DATA_BLOCK "ZEN_Bef"
{ S7_Optimized_Access := 'FALSE' }
VERSION : 0.1
NON_RETAIN
   STRUCT
      ZEN_Quit_BF : Bool;   // UV BG - SPS Quit
      ZEN_Bed_Sperre_BF : Bool;   // UV BG Bedienstelle - Bedienung sperren
      ZEN_Bed_Frg_BF : Bool;   // UV BG Bedienstelle - Bedienung freigeben
      ZEN_ObjS_unscharf_BF : Bool;   // Betriebsgebäude - Objektschutz - Freischaltung
      ZEN_ObjS_scharf_BF : Bool;   // Betriebsgebäude - Objektschutz - Scharfschaltung
      ZEN_GWA_RST_BF : Bool;   // Gaswarnanlagen - Fern-Reset
      ZEN_IEC_RST_BF : Bool;   // IEC-Stack Reset
      ZEN_Res_DB101_0_7 : Bool;   // Reserve
      Biocos1_BA_SU_BF : Bool;   // Steuerung Biocos 1 - Betriebsart - Schaltuhrbetrieb - Befehl
      Biocos1_BA_P1_BF : Bool;   // Steuerung Biocos 1 - Betriebsart - Parametersatz 1 - Befehl
      Biocos1_BA_P2_BF : Bool;   // Steuerung Biocos 1 - Betriebsart - Parametersatz 2 - Befehl
      Biocos1_BA_Aus_BF : Bool;   // Steuerung Biocos 1 - Betriebsart - Aus - Befehl
      Biocos1_Auto_Bel_O2_Ein_BF : Bool;   // Steuerung Biocos 1 - Automatik - Belüftung nach O2-Gehalt - Befehl Ein
      Biocos1_Auto_Bel_O2_Aus_BF : Bool;   // Steuerung Biocos 1 - Automatik - Belüftung nach O2-Gehalt - Befehl Aus
      Biocos1_Auto_UeSS_Menge_Ein_BF : Bool;   // Steuerung Biocos 1 - Automatik - ÜSS-Abzug nach Menge - Befehl Ein
      Biocos1_Auto_UeSS_Menge_Aus_BF : Bool;   // Steuerung Biocos 1 - Automatik - ÜSS-Abzug nach Menge - Befehl Aus
      Biocos2_BA_SU_BF : Bool;   // Steuerung Biocos 2 - Betriebsart - Schaltuhrbetrieb - Befehl
      Biocos2_BA_P1_BF : Bool;   // Steuerung Biocos 2 - Betriebsart - Parametersatz 1 - Befehl
      Biocos2_BA_P2_BF : Bool;   // Steuerung Biocos 2 - Betriebsart - Parametersatz 2 - Befehl
      Biocos2_BA_Aus_BF : Bool;   // Steuerung Biocos 2 - Betriebsart - Aus - Befehl
      Biocos2_Auto_Bel_O2_Ein_BF : Bool;   // Steuerung Biocos 2 - Automatik - Belüftung nach O2-Gehalt - Befehl Ein
      Biocos2_Auto_Bel_O2_Aus_BF : Bool;   // Steuerung Biocos 2 - Automatik - Belüftung nach O2-Gehalt - Befehl Aus
      Biocos2_Auto_UeSS_Menge_Ein_BF : Bool;   // Steuerung Biocos 2 - Automatik - ÜSS-Abzug nach Menge - Befehl Ein
      Biocos2_Auto_UeSS_Menge_Aus_BF : Bool;   // Steuerung Biocos 2 - Automatik - ÜSS-Abzug nach Menge - Befehl Aus
      Zulauf_PW_BA_Auto_BF : Bool;   // Steuerung Zulauf/Freigabe Pumpwerke - Betriebsart - Automatik - Befehl
      Zulauf_PW_BA_Aus_BF : Bool;   // Steuerung Zulauf/Freigabe Pumpwerke - Betriebsart - Aus - Befehl
      Zulauf_PW_BA_EFrg_Ein_BF : Bool;   // Steuerung Zulauf/Freigabe Pumpwerke - Betriebsart - einzelne Freigabe zuschalten - Befehl
      Zulauf_PW_BA_EFrg_Aus_BF : Bool;   // Steuerung Zulauf/Freigabe Pumpwerke - Betriebsart - einzelne Freigabe abschalten - Befehl
      Zulauf_PW_BA_SFrg_Ein_BF : Bool;   // Steuerung Zulauf/Freigabe Pumpwerke - Betriebsart - alle Freigaben zuschalten - Befehl
      Zulauf_PW_BA_SFrg_Aus_BF : Bool;   // Steuerung Zulauf/Freigabe Pumpwerke - Betriebsart - alle Freigaben abschalten - Befehl
      ZEN_Res_DB101_3_6 : Bool;   // Reserve
      ZEN_Res_DB101_3_7 : Bool;   // Reserve
      Schlamm_TW_BA_Auto_BF : Bool;   // Steuerung Trübwasserpumpwerk - Betriebsart - Automatik - Befehl
      Schlamm_TW_BA_Aus_BF : Bool;   // Steuerung Trübwasserpumpwerk - Betriebsart - Aus - Befehl
      ZEN_Res_DB101_4_2 : Bool;   // Reserve
      ZEN_Res_DB101_4_3 : Bool;   // Reserve
      ZEN_Res_DB101_4_4 : Bool;   // Reserve
      ZEN_Res_DB101_4_5 : Bool;   // Reserve
      ZEN_Res_DB101_4_6 : Bool;   // Reserve
      ZEN_Res_DB101_4_7 : Bool;   // Reserve
      Schlamm_Besch_BA_Auto_BF : Bool;   // Steuerung Beschickung Schlammbeete - Betriebsart - Automatik - Befehl
      Schlamm_Besch_BA_Aus_BF : Bool;   // Steuerung Beschickung Schlammbeete - Betriebsart - Aus - Befehl
      ZEN_Res_DB101_5_2 : Bool;   // Reserve
      ZEN_Res_DB101_5_3 : Bool;   // Reserve
      ZEN_Res_DB101_5_4 : Bool;   // Reserve
      ZEN_Res_DB101_5_5 : Bool;   // Reserve
      ZEN_Res_DB101_5_6 : Bool;   // Reserve
      ZEN_Res_DB101_5_7 : Bool;   // Reserve
      PO4_Elim_BA_Auto_BF : Bool;   // Steuerung PO4-Elimination - Betriebsart - Automatik - Befehl
      PO4_Elim_BA_Hand_BF : Bool;   // Steuerung PO4-Elimination - Betriebsart - Handvorgabe - Befehl
      PO4_Elim_BA_Aus_BF : Bool;   // Steuerung PO4-Elimination - Betriebsart - Aus - Befehl
      PO4_Elim_DF_RST_BF : Bool;   // Steuerung PO4-Elimination - Menge Fällmittel - Reset - Befehl
      ZEN_Res_DB101_6_4 : Bool;   // Reserve
      ZEN_Res_DB101_6_5 : Bool;   // Reserve
      ZEN_Res_DB101_6_6 : Bool;   // Reserve
      ZEN_Res_DB101_6_7 : Bool;   // Reserve
      Biocos1_BA_O2_Reg_FW_BF : Bool;   // Steuerung Biocos 1 - Betriebsart O2-Regler - Festwert - Befehl
      Biocos1_BA_O2_Reg_Auto_BF : Bool;   // Steuerung Biocos 1 - Betriebsart O2-Regler - Automatik - Befehl
      ZEN_Res_DB101_7_2 : Bool;   // Reserve
      ZEN_Res_DB101_7_3 : Bool;   // Reserve
      ZEN_Res_DB101_7_4 : Bool;   // Reserve
      ZEN_Res_DB101_7_5 : Bool;   // Reserve
      ZEN_Res_DB101_7_6 : Bool;   // Reserve
      ZEN_Res_DB101_7_7 : Bool;   // Reserve
      Biocos2_BA_O2_Reg_FW_BF : Bool;   // Steuerung Biocos 2 - Betriebsart O2-Regler - Festwert - Befehl
      Biocos2_BA_O2_Reg_Auto_BF : Bool;   // Steuerung Biocos 2 - Betriebsart O2-Regler - Automatik - Befehl
      ZEN_Res_DB101_8_2 : Bool;   // Reserve
      ZEN_Res_DB101_8_3 : Bool;   // Reserve
      ZEN_Res_DB101_8_4 : Bool;   // Reserve
      ZEN_Res_DB101_8_5 : Bool;   // Reserve
      ZEN_Res_DB101_8_6 : Bool;   // Reserve
      ZEN_Res_DB101_8_7 : Bool;   // Reserve
      RES : Array[0..9] of Byte;
   END_STRUCT;


BEGIN

END_DATA_BLOCK

DATA_BLOCK "IDB_SL_Org_ASDU_1"
{ S7_Optimized_Access := 'FALSE' }
AUTHOR : SIE_GST
FAMILY : S7_IEC
VERSION : 0.1
"SL_Org_Asdu_1"

BEGIN

END_DATA_BLOCK

DATA_BLOCK "IDB_MA_Org_ASDU_1"
{ S7_Optimized_Access := 'FALSE' }
AUTHOR : SIE_GST
FAMILY : S7_IEC
VERSION : 0.1
"MA_Org_Asdu_n"

BEGIN

END_DATA_BLOCK

DATA_BLOCK "DB_IEC_PW_Image"
{ S7_Optimized_Access := 'FALSE' }
VERSION : 0.1
   STRUCT
      FW_APW_Oeb_KB : "T_IEC_PW_Image";   // Oebisfelde APW Krumme Breite
      FW_APW_BrR_DM : "T_IEC_PW_Image";   // Breitenrode APW Denkmal
      FW_APW_Oeb_Tu : "T_IEC_PW_Image";   // Oebisfelde APW Tunnel
      FW_APW_Oeb_KS : "T_IEC_PW_Image";   // Oebisfelde APW Klötzer Str.
      FW_APW_Oeb_PG : "T_IEC_PW_Image";   // Oebisfelde APW Papengraben
      FW_APW_Oeb_LW : "T_IEC_PW_Image";   // Oebisfelde APW Lehmweg
      FW_APW_GeD_WG : "T_IEC_PW_Image";   // Gehrendorf APW Wiesengrund
      FW_APW_GeD_AA : "T_IEC_PW_Image";   // Gehrendorf APW An der Aller
      FW_APW_WaD : "T_IEC_PW_Image";   // Wassensdorf APW
      FW_APW_WeD : "T_IEC_PW_Image";   // Weddendorf APW
      FW_APW_NiD : "T_IEC_PW_Image";   // Niendorf APW
      FW_APW_LoS : "T_IEC_PW_Image";   // Lockstedt APW
      FW_APW_Oeb_Ge : "T_IEC_PW_Image";   // Oebisfelde APW Gewerbe
      FW_APW_BuH : "T_IEC_PW_Image";   // Buchhorst APW
      FW_APW_BrR_TS : "T_IEC_PW_Image";   // Breitenrode APW Trafostation
   END_STRUCT;


BEGIN

END_DATA_BLOCK

DATA_BLOCK "ZEN_SW"
{ S7_Optimized_Access := 'FALSE' }
VERSION : 0.1
   STRUCT
      BB_Auto_GeblW_ZZ_SW : DInt;   // Steuerung Belüftung - Automatik - Zykluszeit Gebläsetausch
      Biocos1_Auto_Bel_O2_Int_SW : Real;   // Steuerung Biocos 1 - Automatik - Sollwert O2-Gehalt am Ende Belüftungsintervall
      Biocos1_Auto_Bel_O2_min_SW : Real;   // Steuerung Biocos 1 - Automatik - Grenzwert Sauerstoffeintrag min. pro Belüftungsphase
      Biocos1_Auto_Bel_O2_Zt_min_SW : DInt;   // Steuerung Biocos 1 - Automatik - Mindestbelüftungsdauer pro Intervall
      Biocos1_Auto_UeSS_Zyk_SW : DInt;   // Steuerung Biocos 1 - Automatik - ÜSS-Abzug alle X Zyklen
      Biocos1_Auto_P1_Start_SW : DInt;   // Steuerung Biocos 1 - Automatik - Startzeit Parametersatz 1
      Biocos1_Auto_P2_Start_SW : DInt;   // Steuerung Biocos 1 - Automatik - Startzeit Parametersatz 2
      Biocos1_Auto_U_Zt_P1_SW : DInt;   // Steuerung Biocos 1 - Automatik - Sollwert U-Phase - Parametersatz 1
      Biocos1_Auto_V_Zt_P1_SW : DInt;   // Steuerung Biocos 1 - Automatik - Sollwert V-Phase - Parametersatz 1
      Biocos1_Auto_Bel_Vz_P1_SW : DInt;   // Steuerung Biocos 1 - Automatik - Sollwert Verzögerungszeit Belüftungsphase - Parametersatz 1
      Biocos1_Auto_Bel_Int_P1_SW : DInt;   // Steuerung Biocos 1 - Automatik - Sollwert Anzahl Belüftungsintervalle - Parametersatz 1
      Biocos1_Auto_Bel_Int_Zt_P1_SW : DInt;   // Steuerung Biocos 1 - Automatik - Sollwert Belüftungsdauer (fest) pro Intervall - Parametersatz 1
      Biocos1_Auto_UeSS_Zt_P1_SW : DInt;   // Steuerung Biocos 1 - Automatik - Sollwert ÜSS-Abzug Dauer - Parametersatz 1
      Biocos1_Auto_UeSS_Df_P1_SW : Real;   // Steuerung Biocos 1 - Automatik - Sollwert ÜSS-Abzug Menge - Parametersatz 1
      Biocos1_Auto_SR1_Zt_P1_SW : DInt;   // Steuerung Biocos 1 - Automatik - Sollwert Dauer Schlammrückführung SU-Becken 1 - Parametersatz 1
      Biocos1_Auto_SR2_Zt_P1_SW : DInt;   // Steuerung Biocos 1 - Automatik - Sollwert Dauer Schlammrückführung SU-Becken 2 - Parametersatz 1
      Biocos1_Auto_U_Zt_P2_SW : DInt;   // Steuerung Biocos 1 - Automatik - Sollwert U-Phase - Parametersatz 2
      Biocos1_Auto_V_Zt_P2_SW : DInt;   // Steuerung Biocos 1 - Automatik - Sollwert V-Phase - Parametersatz 2
      Biocos1_Auto_Bel_Vz_P2_SW : DInt;   // Steuerung Biocos 1 - Automatik - Sollwert Verzögerungszeit Belüftungsphase - Parametersatz 2
      Biocos1_Auto_Bel_Int_P2_SW : DInt;   // Steuerung Biocos 1 - Automatik - Sollwert Anzahl Belüftungsintervalle - Parametersatz 2
      Biocos1_Auto_Bel_Int_Zt_P2_SW : DInt;   // Steuerung Biocos 1 - Automatik - Sollwert Belüftungsdauer (fest) pro Intervall - Parametersatz 2
      Biocos1_Auto_UeSS_Zt_P2_SW : DInt;   // Steuerung Biocos 1 - Automatik - Sollwert ÜSS-Abzug Dauer - Parametersatz 2
      Biocos1_Auto_UeSS_Df_P2_SW : Real;   // Steuerung Biocos 1 - Automatik - Sollwert ÜSS-Abzug Menge - Parametersatz 2
      Biocos1_Auto_SR1_Zt_P2_SW : DInt;   // Steuerung Biocos 1 - Automatik - Sollwert Dauer Schlammrückführung SU-Becken 1 - Parametersatz 2
      Biocos1_Auto_SR2_Zt_P2_SW : DInt;   // Steuerung Biocos 1 - Automatik - Sollwert Dauer Schlammrückführung SU-Becken 2 - Parametersatz 2
      Biocos2_Auto_Bel_O2_Int_SW : Real;   // Steuerung Biocos 2 - Automatik - Sollwert O2-Gehalt am Ende Belüftungsintervall
      Biocos2_Auto_Bel_O2_min_SW : Real;   // Steuerung Biocos 2 - Automatik - Grenzwert Sauerstoffeintrag min. pro Belüftungsphase
      Biocos2_Auto_Bel_O2_Zt_min_SW : DInt;   // Steuerung Biocos 2 - Automatik - Mindestbelüftungsdauer pro Intervall
      Biocos2_Auto_UeSS_Zyk_SW : DInt;   // Steuerung Biocos 2 - Automatik - ÜSS-Abzug alle X Zyklen
      Biocos2_Auto_P1_Start_SW : DInt;   // Steuerung Biocos 2 - Automatik - Startzeit Parametersatz 1
      Biocos2_Auto_P2_Start_SW : DInt;   // Steuerung Biocos 2 - Automatik - Startzeit Parametersatz 2
      Biocos2_Auto_U_Zt_P1_SW : DInt;   // Steuerung Biocos 2 - Automatik - Sollwert U-Phase - Parametersatz 1
      Biocos2_Auto_V_Zt_P1_SW : DInt;   // Steuerung Biocos 2 - Automatik - Sollwert V-Phase - Parametersatz 1
      Biocos2_Auto_Bel_Vz_P1_SW : DInt;   // Steuerung Biocos 2 - Automatik - Sollwert Verzögerungszeit Belüftungsphase - Parametersatz 1
      Biocos2_Auto_Bel_Int_P1_SW : DInt;   // Steuerung Biocos 2 - Automatik - Sollwert Anzahl Belüftungsintervalle - Parametersatz 1
      Biocos2_Auto_Bel_Int_Zt_P1_SW : DInt;   // Steuerung Biocos 2 - Automatik - Sollwert Belüftungsdauer (fest) pro Intervall - Parametersatz 1
      Biocos2_Auto_UeSS_Zt_P1_SW : DInt;   // Steuerung Biocos 2 - Automatik - Sollwert ÜSS-Abzug Dauer - Parametersatz 1
      Biocos2_Auto_UeSS_Df_P1_SW : Real;   // Steuerung Biocos 2 - Automatik - Sollwert ÜSS-Abzug Menge - Parametersatz 1
      Biocos2_Auto_SR1_Zt_P1_SW : DInt;   // Steuerung Biocos 2 - Automatik - Sollwert Dauer Schlammrückführung SU-Becken 1 - Parametersatz 1
      Biocos2_Auto_SR2_Zt_P1_SW : DInt;   // Steuerung Biocos 2 - Automatik - Sollwert Dauer Schlammrückführung SU-Becken 2 - Parametersatz 1
      Biocos2_Auto_U_Zt_P2_SW : DInt;   // Steuerung Biocos 2 - Automatik - Sollwert U-Phase - Parametersatz 2
      Biocos2_Auto_V_Zt_P2_SW : DInt;   // Steuerung Biocos 2 - Automatik - Sollwert V-Phase - Parametersatz 2
      Biocos2_Auto_Bel_Vz_P2_SW : DInt;   // Steuerung Biocos 2 - Automatik - Sollwert Verzögerungszeit Belüftungsphase - Parametersatz 2
      Biocos2_Auto_Bel_Int_P2_SW : DInt;   // Steuerung Biocos 2 - Automatik - Sollwert Anzahl Belüftungsintervalle - Parametersatz 2
      Biocos2_Auto_Bel_Int_Zt_P2_SW : DInt;   // Steuerung Biocos 2 - Automatik - Sollwert Belüftungsdauer (fest) pro Intervall - Parametersatz 2
      Biocos2_Auto_UeSS_Zt_P2_SW : DInt;   // Steuerung Biocos 2 - Automatik - Sollwert ÜSS-Abzug Dauer - Parametersatz 2
      Biocos2_Auto_UeSS_Df_P2_SW : Real;   // Steuerung Biocos 2 - Automatik - Sollwert ÜSS-Abzug Menge - Parametersatz 2
      Biocos2_Auto_SR1_Zt_P2_SW : DInt;   // Steuerung Biocos 2 - Automatik - Sollwert Dauer Schlammrückführung SU-Becken 1 - Parametersatz 2
      Biocos2_Auto_SR2_Zt_P2_SW : DInt;   // Steuerung Biocos 2 - Automatik - Sollwert Dauer Schlammrückführung SU-Becken 2 - Parametersatz 2
      Zulauf_PW_Auto_DF_max_SW : Real;   // Steuerung Zulauf/Freigabe Pumpwerke - Grenzwert max. Durchflußmenge durch die KA
      Zulauf_PW_Auto_Niv_max_SW : Real;   // Steuerung Zulauf/Freigabe Pumpwerke - Niveau Vorlageschacht Zulauf - alle Freigaben ext. PW abschalten
      Zulauf_PW_Auto_Niv_AS_SW : Real;   // Steuerung Zulauf/Freigabe Pumpwerke - Niveau Vorlageschacht Zulauf - Freigabe ext. PW abschalten
      Zulauf_PW_Auto_Niv_ZS_SW : Real;   // Steuerung Zulauf/Freigabe Pumpwerke - Niveau Vorlageschacht Zulauf - Freigabe ext. PW zuschalten
      Zulauf_PW_Auto_Niv_min_SW : Real;   // Steuerung Zulauf/Freigabe Pumpwerke - Niveau Vorlageschacht Zulauf - alle Freigaben ext. PW zuschalten
      Zulauf_PW_Auto_Zyk_SW : DInt;   // Steuerung Zulauf/Freigabe Pumpwerke - Zykluszeit Zu-/Abschaltung Pumpwerke
      Schlamm_TW_Auto_Frg_Zt_Ein_SW : DInt;   // Steuerung Trübwasserpumpwerk - Startzeit Freigabe Abzug
      Schlamm_TW_Auto_Frg_Zt_Aus_SW : DInt;   // Steuerung Trübwasserpumpwerk - Endzeit Freigabe Abzug
      Schlamm_TW_Auto_Niv_2P_Ein_SW : Real;   // Steuerung Trübwasserpumpwerk - Niveau Trübwasserschacht - Abpumpen 2 Pumpen Ein
      Schlamm_TW_Auto_Niv_1P_Ein_SW : Real;   // Steuerung Trübwasserpumpwerk - Niveau Trübwasserschacht - Abpumpen 1 Pumpe Ein
      Schlamm_TW_Auto_Niv_Aus_SW : Real;   // Steuerung Trübwasserpumpwerk - Niveau Trübwasserschacht - Abpumpen Aus
      Schlamm_Besch_Auto_Menge_SW : DInt;   // Steuerung Beschickung Schlammbeete - Menge Beschickung - Sollwert
      Schlamm_Besch_Auto_Zt_max_SW : DInt;   // Steuerung Beschickung Schlammbeete - Überwachungszeit
      PO4_Elim_BA_Hand_SW : Real;   // Steuerung PO4-Elimination - Betriebsart Hand - Menge Fällmittel - Sollwert
      Biocos1_Auto_Bel_O2_Reg_FW : Real;   // Steuerung Biocos 1 - Automatik O2-Regler - Vorgabe Festwert Blockdrehzahl für Ansteuerung Gebläse
      Biocos1_Auto_Bel_O2_Reg_GW_max : Real;   // Steuerung Biocos 1 - Automatik O2-Regler - Sollwert O2-Gehalt max -> Abschaltung Gebläse
      Biocos1_Auto_Bel_O2_Reg_GW_ein : Real;   // Steuerung Biocos 1 - Automatik O2-Regler - Sollwert O2-Gehalt min -> Einschaltung Gebläse
      Biocos1_Auto_Bel_O2_Reg_SW_max : Real;   // Steuerung Biocos 1 - Automatik O2-Regler - Sollwert O2-Gehalt max -> Gebläse auf min-Drehzahl
      Biocos1_Auto_Bel_O2_Reg_SW_min : Real;   // Steuerung Biocos 1 - Automatik O2-Regler - Sollwert O2-Gehalt min -> Gebläse auf max-Drehzahl
      Biocos1_Auto_Bel_O2_Reg_DZ_max : Real;   // Steuerung Biocos 1 - Automatik O2-Regler - Sollwert Blockdrehzahl max bei O2 min
      Biocos1_Auto_Bel_O2_Reg_DZ_min : Real;   // Steuerung Biocos 1 - Automatik O2-Regler - Sollwert Blockdrehzahl min bei O2 max
      Biocos2_Auto_Bel_O2_Reg_FW : Real;   // Steuerung Biocos 2 - Automatik O2-Regler - Vorgabe Festwert Blockdrehzahl für Ansteuerung Gebläse
      Biocos2_Auto_Bel_O2_Reg_GW_max : Real;   // Steuerung Biocos 2 - Automatik O2-Regler - Sollwert O2-Gehalt max -> Abschaltung Gebläse
      Biocos2_Auto_Bel_O2_Reg_GW_ein : Real;   // Steuerung Biocos 2 - Automatik O2-Regler - Sollwert O2-Gehalt min -> Einschaltung Gebläse
      Biocos2_Auto_Bel_O2_Reg_SW_max : Real;   // Steuerung Biocos 2 - Automatik O2-Regler - Sollwert O2-Gehalt max -> Gebläse auf min-Drehzahl
      Biocos2_Auto_Bel_O2_Reg_SW_min : Real;   // Steuerung Biocos 2 - Automatik O2-Regler - Sollwert O2-Gehalt min -> Gebläse auf max-Drehzahl
      Biocos2_Auto_Bel_O2_Reg_DZ_max : Real;   // Steuerung Biocos 2 - Automatik O2-Regler - Sollwert Blockdrehzahl max bei O2 min
      Biocos2_Auto_Bel_O2_Reg_DZ_min : Real;   // Steuerung Biocos 2 - Automatik O2-Regler - Sollwert Blockdrehzahl min bei O2 max
      RES : Array[0..9] of Byte;
   END_STRUCT;


BEGIN
   BB_Auto_GeblW_ZZ_SW := 24;
   Biocos1_Auto_Bel_O2_Int_SW := 2.0;
   Biocos1_Auto_Bel_O2_min_SW := 0.5;
   Biocos1_Auto_Bel_O2_Zt_min_SW := 300;
   Biocos1_Auto_UeSS_Zyk_SW := 1;
   Biocos1_Auto_P1_Start_SW := 8;
   Biocos1_Auto_P2_Start_SW := 0;
   Biocos1_Auto_U_Zt_P1_SW := 15;
   Biocos1_Auto_V_Zt_P1_SW := 45;
   Biocos1_Auto_Bel_Vz_P1_SW := 60;
   Biocos1_Auto_Bel_Int_P1_SW := 3;
   Biocos1_Auto_Bel_Int_Zt_P1_SW := 300;
   Biocos1_Auto_UeSS_Zt_P1_SW := 8;
   Biocos1_Auto_UeSS_Df_P1_SW := 1.0;
   Biocos1_Auto_SR1_Zt_P1_SW := 3;
   Biocos1_Auto_SR2_Zt_P1_SW := 3;
   Biocos1_Auto_U_Zt_P2_SW := 15;
   Biocos1_Auto_V_Zt_P2_SW := 75;
   Biocos1_Auto_Bel_Vz_P2_SW := 240;
   Biocos1_Auto_Bel_Int_P2_SW := 3;
   Biocos1_Auto_Bel_Int_Zt_P2_SW := 300;
   Biocos1_Auto_UeSS_Zt_P2_SW := 8;
   Biocos1_Auto_UeSS_Df_P2_SW := 4.0;
   Biocos1_Auto_SR1_Zt_P2_SW := 3;
   Biocos1_Auto_SR2_Zt_P2_SW := 3;
   Biocos2_Auto_Bel_O2_Int_SW := 2.0;
   Biocos2_Auto_Bel_O2_min_SW := 1.5;
   Biocos2_Auto_Bel_O2_Zt_min_SW := 300;
   Biocos2_Auto_UeSS_Zyk_SW := 1;
   Biocos2_Auto_P1_Start_SW := 8;
   Biocos2_Auto_P2_Start_SW := 0;
   Biocos2_Auto_U_Zt_P1_SW := 15;
   Biocos2_Auto_V_Zt_P1_SW := 45;
   Biocos2_Auto_Bel_Vz_P1_SW := 60;
   Biocos2_Auto_Bel_Int_P1_SW := 4;
   Biocos2_Auto_Bel_Int_Zt_P1_SW := 300;
   Biocos2_Auto_UeSS_Zt_P1_SW := 0;
   Biocos2_Auto_UeSS_Df_P1_SW := 0.0;
   Biocos2_Auto_SR1_Zt_P1_SW := 3;
   Biocos2_Auto_SR2_Zt_P1_SW := 3;
   Biocos2_Auto_U_Zt_P2_SW := 15;
   Biocos2_Auto_V_Zt_P2_SW := 75;
   Biocos2_Auto_Bel_Vz_P2_SW := 240;
   Biocos2_Auto_Bel_Int_P2_SW := 3;
   Biocos2_Auto_Bel_Int_Zt_P2_SW := 300;
   Biocos2_Auto_UeSS_Zt_P2_SW := 8;
   Biocos2_Auto_UeSS_Df_P2_SW := 3.5;
   Biocos2_Auto_SR1_Zt_P2_SW := 3;
   Biocos2_Auto_SR2_Zt_P2_SW := 3;
   Zulauf_PW_Auto_DF_max_SW := 50.0;
   Zulauf_PW_Auto_Niv_max_SW := 90.0;
   Zulauf_PW_Auto_Niv_AS_SW := 80.0;
   Zulauf_PW_Auto_Niv_ZS_SW := 60.0;
   Zulauf_PW_Auto_Niv_min_SW := 60.0;
   Zulauf_PW_Auto_Zyk_SW := 60;
   Schlamm_TW_Auto_Frg_Zt_Ein_SW := 8;
   Schlamm_TW_Auto_Frg_Zt_Aus_SW := 8;
   Schlamm_TW_Auto_Niv_2P_Ein_SW := 90.0;
   Schlamm_TW_Auto_Niv_1P_Ein_SW := 45.0;
   Schlamm_TW_Auto_Niv_Aus_SW := 15.0;
   Schlamm_Besch_Auto_Menge_SW := 50;
   Schlamm_Besch_Auto_Zt_max_SW := 70;
   PO4_Elim_BA_Hand_SW := 2.0;
   Biocos1_Auto_Bel_O2_Reg_FW := 6500.0;
   Biocos1_Auto_Bel_O2_Reg_GW_max := 4.0;
   Biocos1_Auto_Bel_O2_Reg_GW_ein := 1.6;
   Biocos1_Auto_Bel_O2_Reg_SW_max := 2.5;
   Biocos1_Auto_Bel_O2_Reg_SW_min := 1.5;
   Biocos1_Auto_Bel_O2_Reg_DZ_max := 8000.0;
   Biocos1_Auto_Bel_O2_Reg_DZ_min := 3000.0;
   Biocos2_Auto_Bel_O2_Reg_FW := 6500.0;
   Biocos2_Auto_Bel_O2_Reg_GW_max := 4.0;
   Biocos2_Auto_Bel_O2_Reg_GW_ein := 1.6;
   Biocos2_Auto_Bel_O2_Reg_SW_max := 2.5;
   Biocos2_Auto_Bel_O2_Reg_SW_min := 1.5;
   Biocos2_Auto_Bel_O2_Reg_DZ_max := 8000.0;
   Biocos2_Auto_Bel_O2_Reg_DZ_min := 3000.0;
   RES[0] := 16#00;
   RES[1] := 16#00;
   RES[2] := 16#00;
   RES[3] := 16#00;
   RES[4] := 16#00;
   RES[5] := 16#00;
   RES[6] := 16#00;
   RES[7] := 16#00;
   RES[8] := 16#00;
   RES[9] := 16#00;

END_DATA_BLOCK

DATA_BLOCK "DB80_Peri_EA"
{ S7_Optimized_Access := 'FALSE' }
VERSION : 0.1
NON_RETAIN
   STRUCT
      Zulauf_DosP { ExternalAccessible := 'False'; ExternalVisible := 'False'; ExternalWritable := 'False'} : "T_EA_FU_CIM_DP";
      PO4_HALA_SC : "T_EA_HALA_SC";
      Kaeser_G1 : "T_EA_KAESER";
      Kaeser_G2 : "T_EA_KAESER";
      Kaeser_G3 : "T_EA_KAESER";
      end { ExternalAccessible := 'False'; ExternalVisible := 'False'; ExternalWritable := 'False'} : Bool;
   END_STRUCT;


BEGIN
   Zulauf_DosP.E.STW.ActRemoteAccess := FALSE;
   Zulauf_DosP.E.STW.ActDeaerating := FALSE;
   Zulauf_DosP.E.STW.ActAnalogMode := TRUE;
   Zulauf_DosP.E.STW.ActTimerMode := FALSE;
   Zulauf_DosP.E.STW.ActSlowMode := FALSE;
   Zulauf_DosP.E.STW.ActVelocity := FALSE;
   Zulauf_DosP.E.STW.Res0_6 := FALSE;
   Zulauf_DosP.E.STW.Res0_7 := FALSE;
   Zulauf_DosP.E.STW.ActAutoDeaeratingEnable := FALSE;
   Zulauf_DosP.E.STW.ActFlowControlEnable := FALSE;
   Zulauf_DosP.E.STW.ActProfiWatchdogEnable := TRUE;
   Zulauf_DosP.E.STW.ActAutoFlowAdaptEnable := FALSE;
   Zulauf_DosP.E.STW.ActPulseMemoryEnable := FALSE;
   Zulauf_DosP.E.STW.Res1_5 := FALSE;
   Zulauf_DosP.E.STW.Res1_6 := FALSE;
   Zulauf_DosP.E.STW.Res1_7 := FALSE;
   Zulauf_DosP.E.STW.ResetFaultAck := FALSE;
   Zulauf_DosP.E.STW.PulseAck := FALSE;
   Zulauf_DosP.E.STW.ResetVolumeCounterAck := FALSE;
   Zulauf_DosP.E.STW.SetRTCAck := FALSE;
   Zulauf_DosP.E.STW.Res2_4 := FALSE;
   Zulauf_DosP.E.STW.Res2_5 := FALSE;
   Zulauf_DosP.E.STW.Res2_6 := FALSE;
   Zulauf_DosP.E.STW.Res2_7 := FALSE;
   Zulauf_DosP.E.STW.Dosierung := FALSE;
   Zulauf_DosP.E.STW.Warning := FALSE;
   Zulauf_DosP.E.STW.Fault := FALSE;
   Zulauf_DosP.E.STW.BusControlLocallyEnabled := TRUE;
   Zulauf_DosP.E.STW.Res3_4 := FALSE;
   Zulauf_DosP.E.STW.Res3_5 := FALSE;
   Zulauf_DosP.E.STW.Res3_6 := FALSE;
   Zulauf_DosP.E.STW.Res3_7 := FALSE;
   Zulauf_DosP.E.STW.ActualStartStop := 16#01;
   Zulauf_DosP.E.STW.ActualOperatingMode := 16#00;
   Zulauf_DosP.E.FltCode := 16#00;
   Zulauf_DosP.E.WrnCode := 16#00;
   Zulauf_DosP.E.WrnBits := 16#0000;
   Zulauf_DosP.E.DosingCapacityReference := 0.0;
   Zulauf_DosP.E.MeasuredDosingCapacity := 0.0;
   Zulauf_DosP.E.MeasuredPressure := 1.0;
   Zulauf_DosP.E.VolumeTotal := 0.422;
   Zulauf_DosP.A.RemoteAccessReq := FALSE;
   Zulauf_DosP.A.Deaerating := FALSE;
   Zulauf_DosP.A.AnalogMode := FALSE;
   Zulauf_DosP.A.TimerMode := FALSE;
   Zulauf_DosP.A.SlowMode := FALSE;
   Zulauf_DosP.A.Velocity := FALSE;
   Zulauf_DosP.A.Res0_6 := FALSE;
   Zulauf_DosP.A.Res0_7 := FALSE;
   Zulauf_DosP.A.AutoDeaeratingEnable := FALSE;
   Zulauf_DosP.A.FlowControlEnable := FALSE;
   Zulauf_DosP.A.ProfiWatchdogEnable := FALSE;
   Zulauf_DosP.A.AutoFlowAdaptEnable := FALSE;
   Zulauf_DosP.A.PulseMemoryEnable := FALSE;
   Zulauf_DosP.A.Res1_5 := FALSE;
   Zulauf_DosP.A.Res1_6 := FALSE;
   Zulauf_DosP.A.Res1_7 := FALSE;
   Zulauf_DosP.A.ResetFault := FALSE;
   Zulauf_DosP.A.Pulse := FALSE;
   Zulauf_DosP.A.ResetVolumeCounter := FALSE;
   Zulauf_DosP.A.SetRTC := FALSE;
   Zulauf_DosP.A.Res2_4 := FALSE;
   Zulauf_DosP.A.Res2_5 := FALSE;
   Zulauf_DosP.A.Res2_6 := FALSE;
   Zulauf_DosP.A.Res2_7 := FALSE;
   Zulauf_DosP.A.ReqStartStop := 16#01;
   Zulauf_DosP.A.OperatingMode := 16#00;
   Zulauf_DosP.A.SetSetpointManual := 0.0;
   Zulauf_DosP.A_DP.Data[0] := 16#00;
   Zulauf_DosP.A_DP.Data[1] := 16#00;
   Zulauf_DosP.A_DP.Data[2] := 16#00;
   Zulauf_DosP.A_DP.Data[3] := 16#00;
   Zulauf_DosP.A_DP.Data[4] := 16#00;
   Zulauf_DosP.A_DP.Res := 16#00;
   PO4_HALA_SC.E.DEV_WARNINGS."MODBUS ADDRESS" := FALSE;
   PO4_HALA_SC.E.DEV_WARNINGS."PROBE SERVICE" := FALSE;
   PO4_HALA_SC.E.DEV_WARNINGS."SENSOR MISSING" := FALSE;
   PO4_HALA_SC.E.DEV_WARNINGS."SENSOR FAIL" := FALSE;
   PO4_HALA_SC.E.DEV_WARNINGS."SENSOR EXCEPTION" := FALSE;
   PO4_HALA_SC.E.DEV_WARNINGS."CH1: FALLBACK STRATEGY" := FALSE;
   PO4_HALA_SC.E.DEV_WARNINGS."CH2: FALLBACK STRATEGY" := FALSE;
   PO4_HALA_SC.E.DEV_WARNINGS."ANALOGUE INPUT1 FAULTY" := FALSE;
   PO4_HALA_SC.E.DEV_WARNINGS."ANALOGUE INPUT2 FAULTY" := FALSE;
   PO4_HALA_SC.E.DEV_WARNINGS."ANALOGUE INPUT3 FAULTY" := FALSE;
   PO4_HALA_SC.E.DEV_WARNINGS."ANALOGUE INPUT4 FAULTY" := FALSE;
   PO4_HALA_SC.E.DEV_ERRORS."RTC MISSING" := FALSE;
   PO4_HALA_SC.E.DEV_ERRORS."RTC CRC" := FALSE;
   PO4_HALA_SC.E.DEV_ERRORS."CHECK CONFIG" := FALSE;
   PO4_HALA_SC.E.DEV_ERRORS."SYNTAX ERROR" := FALSE;
   PO4_HALA_SC.E.DEV_ERRORS."FORMULA TO LONG" := FALSE;
   PO4_HALA_SC.E.DEV_ERRORS.ARGUMENT := FALSE;
   PO4_HALA_SC.E.DEV_ERRORS."LOGIC FUNCTION" := FALSE;
   PO4_HALA_SC.E.DEV_ERRORS."BOUNDARY FUNCTION" := FALSE;
   PO4_HALA_SC.E.DEV_ERRORS."TOO MANY PROBES" := FALSE;
   PO4_HALA_SC.E.DEV_ERRORS."TOO MANY MEASUREMENTS" := FALSE;
   PO4_HALA_SC.E.DEV_ERRORS."RTC FAILURE" := FALSE;
   PO4_HALA_SC.E.DosP_Anf := 0.0;
   PO4_HALA_SC.E.DF_Dos_SW := 0.0;
   PO4_HALA_SC.E.PO4_akt := 0.0;
   PO4_HALA_SC.A.DF_Zulauf := 12.48366;
   PO4_HALA_SC.A.DF_DosM := 0.0;
   PO4_HALA_SC.A.DF_RS := 0.0;
   PO4_HALA_SC.A.PO4_akt := 2.265022;
   PO4_HALA_SC.A.Res_16 := 0.0;
   PO4_HALA_SC.A.Res_20 := 0.0;
   PO4_HALA_SC.A.Res_24 := 0.0;
   PO4_HALA_SC.A.Res_28 := 0.0;
   end := FALSE;

END_DATA_BLOCK

DATA_BLOCK "DB_IEC_MW_Image"
{ DB_Accessible_From_OPC_UA := 'FALSE' ;
 S7_Optimized_Access := 'FALSE' }
VERSION : 0.1
NON_RETAIN
   STRUCT
      Umwelt_WG { S7_SetPoint := 'False'} : "T_IEC_Sli_MEfl_Img";   // Wetterstation Windgeschwindigkeit
      Umwelt_WR { S7_SetPoint := 'False'} : "T_IEC_Sli_MEfl_Img";   // Wetterstation Windrichtung
      Umwelt_T { S7_SetPoint := 'False'} : "T_IEC_Sli_MEfl_Img";   // Wetterstation Temperatur
      Umwelt_LDr { S7_SetPoint := 'False'} : "T_IEC_Sli_MEfl_Img";   // Wetterstation Luftdruck
      Umwelt_LF { S7_SetPoint := 'False'} : "T_IEC_Sli_MEfl_Img";   // Wetterstation rel.Feuchte
      Umwelt_RM { S7_SetPoint := 'False'} : "T_IEC_Sli_TI_Img";   // Wetterstation Niederschlag
   END_STRUCT;


BEGIN

END_DATA_BLOCK

DATA_BLOCK "DB_IEC_Config"
TITLE = Konfigurationsdaten für IEC-Stack
{ S7_Optimized_Access := 'TRUE' }
VERSION : 0.1
   VAR
      Prm_Line : "T_IEC_LINE_CFG";
      Prm_ASDU : Array[1..16] of "T_IEC_ASDU_CFG";
   END_VAR


BEGIN
   Prm_Line.Reg_Code := DWORD#16#A243_47D1;
   Prm_Line.First_IntDB := 1000;
   Prm_ASDU[1].ASDU_Adr := DINT#25602;
   Prm_ASDU[2].ASDU_Adr := DINT#100_000_401;

END_DATA_BLOCK

DATA_BLOCK "DB90_MW_Mittel"
{ S7_Optimized_Access := 'TRUE' }
VERSION : 0.1
NON_RETAIN
   VAR
      Zulauf_AR_Niv { ExternalAccessible := 'False'; ExternalVisible := 'False'; ExternalWritable := 'False'} : "T_MW_MITTEL";   // Zulauf - Pumpwerk "Alter Rechen" - Niveau
      Zulauf_AR_Temp { ExternalAccessible := 'False'; ExternalVisible := 'False'; ExternalWritable := 'False'} : "T_MW_MITTEL";   // Zulauf - Pumpwerk "Alter Rechen" - Temperatur
      Zulauf_AR_DF { ExternalAccessible := 'False'; ExternalVisible := 'False'; ExternalWritable := 'False'} : "T_MW_MITTEL";   // Zulauf - Pumpwerk "Alter Rechen" - Durchfluss
      BB1_AS1_SS { ExternalAccessible := 'False'; ExternalVisible := 'False'; ExternalWritable := 'False'} : "T_MW_MITTEL";   // Becken 1 - Ablaufschieber 1 - Schieberstellung
      BB1_AS2_SS { ExternalAccessible := 'False'; ExternalVisible := 'False'; ExternalWritable := 'False'} : "T_MW_MITTEL";   // Becken 1 - Ablaufschieber 2 - Schieberstellung
      BB2_AS1_SS { ExternalAccessible := 'False'; ExternalVisible := 'False'; ExternalWritable := 'False'} : "T_MW_MITTEL";   // Becken 2 - Ablaufschieber 1 - Schieberstellung
      BB2_AS2_SS { ExternalAccessible := 'False'; ExternalVisible := 'False'; ExternalWritable := 'False'} : "T_MW_MITTEL";   // Becken 2 - Ablaufschieber 2 - Schieberstellung
      BB1_O2 { ExternalAccessible := 'False'; ExternalVisible := 'False'; ExternalWritable := 'False'} : "T_MW_MITTEL";   // Becken 1 - O2-Gehalt
      BB1_Temp { ExternalAccessible := 'False'; ExternalVisible := 'False'; ExternalWritable := 'False'} : "T_MW_MITTEL";   // Becken 1 - Temperatur
      BB2_O2 { ExternalAccessible := 'False'; ExternalVisible := 'False'; ExternalWritable := 'False'} : "T_MW_MITTEL";   // Becken 2 - O2-Gehalt
      BB2_Temp { ExternalAccessible := 'False'; ExternalVisible := 'False'; ExternalWritable := 'False'} : "T_MW_MITTEL";   // Becken 2 - Temperatur
      BB1_DF { ExternalAccessible := 'False'; ExternalVisible := 'False'; ExternalWritable := 'False'} : "T_MW_MITTEL";   // Becken 1 - Ablauf - Durchfluss
      BB2_DF { ExternalAccessible := 'False'; ExternalVisible := 'False'; ExternalWritable := 'False'} : "T_MW_MITTEL";   // Becken 2 - Ablauf - Durchfluss
      Zulauf_Niv { ExternalAccessible := 'False'; ExternalVisible := 'False'; ExternalWritable := 'False'} : "T_MW_MITTEL";   // Zulauf - Vorlagebehälter - Niveau
      Zulauf_DF { ExternalAccessible := 'False'; ExternalVisible := 'False'; ExternalWritable := 'False'} : "T_MW_MITTEL";   // Zulauf - Rechen - Durchfluss
      Verteiler_pH { ExternalAccessible := 'False'; ExternalVisible := 'False'; ExternalWritable := 'False'} : "T_MW_MITTEL";   // Zulauf - Verteiler - pH-Wert
      Verteiler_O2 { ExternalAccessible := 'False'; ExternalVisible := 'False'; ExternalWritable := 'False'} : "T_MW_MITTEL";   // Zulauf - Verteiler  - O2-Gehalt
      Verteiler_Temp { ExternalAccessible := 'False'; ExternalVisible := 'False'; ExternalWritable := 'False'} : "T_MW_MITTEL";   // Zulauf - Verteiler - Temperatur
      BB_UeSS_DF { ExternalAccessible := 'False'; ExternalVisible := 'False'; ExternalWritable := 'False'} : "T_MW_MITTEL";   // Becken 1+2 - Ablauf ÜSS - Durchfluss
      Ablauf_DF { ExternalAccessible := 'False'; ExternalVisible := 'False'; ExternalWritable := 'False'} : "T_MW_MITTEL";   // Ablauf - Durchfluss
      Ablauf_pH { ExternalAccessible := 'False'; ExternalVisible := 'False'; ExternalWritable := 'False'} : "T_MW_MITTEL";   // Ablauf - pH-Wert
      Ablauf_O2 { ExternalAccessible := 'False'; ExternalVisible := 'False'; ExternalWritable := 'False'} : "T_MW_MITTEL";   // Ablauf - O2-Gehalt
      Ablauf_Temp { ExternalAccessible := 'False'; ExternalVisible := 'False'; ExternalWritable := 'False'} : "T_MW_MITTEL";   // Ablauf - Temperatur
      Schlamm_ED_Niv { ExternalAccessible := 'False'; ExternalVisible := 'False'; ExternalWritable := 'False'} : "T_MW_MITTEL";   // Schlamm - Eindicker - Niveau
      Schlamm_Besch_Niv { ExternalAccessible := 'False'; ExternalVisible := 'False'; ExternalWritable := 'False'} : "T_MW_MITTEL";   // Schlamm - Beschickung - Niveau
      Schlamm_Besch_DF { ExternalAccessible := 'False'; ExternalVisible := 'False'; ExternalWritable := 'False'} : "T_MW_MITTEL";   // Schlamm - Beschickung - Durchfluss
      Truebwasser_Niv { ExternalAccessible := 'False'; ExternalVisible := 'False'; ExternalWritable := 'False'} : "T_MW_MITTEL";   // Trübwasserpumpwerk - Niveau
      Truebwasser_DF { ExternalAccessible := 'False'; ExternalVisible := 'False'; ExternalWritable := 'False'} : "T_MW_MITTEL";   // Trübwasserpumpwerk - Durchfluss
      Zulauf_SF_Niv { ExternalAccessible := 'False'; ExternalVisible := 'False'; ExternalWritable := 'False'} : "T_MW_MITTEL";   // Zulauf - Sandfang - Niveau
      Ablauf_NOx { ExternalAccessible := 'False'; ExternalVisible := 'False'; ExternalWritable := 'False'} : "T_MW_MITTEL";   // Ablauf - Dortmundbrunnen - Nitratmessung
      Ablauf_PO4 { ExternalAccessible := 'False'; ExternalVisible := 'False'; ExternalWritable := 'False'} : "T_MW_MITTEL";   // Ablauf - Dortmundbrunnen - Phosphatmessung
      Umwelt_WG { ExternalAccessible := 'False'; ExternalVisible := 'False'; ExternalWritable := 'False'} : "T_MW_MITTEL";   // Wetterstation - Windgeschwindigkeit
      Umwelt_WR { ExternalAccessible := 'False'; ExternalVisible := 'False'; ExternalWritable := 'False'} : "T_MW_MITTEL";   // Wetterstation - Windrichtung
      Umwelt_LDr { ExternalAccessible := 'False'; ExternalVisible := 'False'; ExternalWritable := 'False'} : "T_MW_MITTEL";   // Wetterstation - Luftdruck
      Umwelt_LF { ExternalAccessible := 'False'; ExternalVisible := 'False'; ExternalWritable := 'False'} : "T_MW_MITTEL";   // Wetterstation - Luftfeuchtigkeit
      Umwelt_T { ExternalAccessible := 'False'; ExternalVisible := 'False'; ExternalWritable := 'False'} : "T_MW_MITTEL";   // Wetterstation - Temperatur
      Ablauf_LF { ExternalAccessible := 'False'; ExternalVisible := 'False'; ExternalWritable := 'False'} : "T_MW_MITTEL";   // Ablauf - Leitfähigkeit
   END_VAR


BEGIN
   Zulauf_AR_Niv.Values[0] := 21.8952;
   Zulauf_AR_Niv.Values[1] := 21.8952;
   Zulauf_AR_Niv.Values[2] := 21.93137;
   Zulauf_AR_Niv.Values[3] := 21.8952;
   Zulauf_AR_Niv.Values[4] := 21.89972;
   Zulauf_AR_Niv.Values[5] := 0.0;
   Zulauf_AR_Niv.Values[6] := 0.0;
   Zulauf_AR_Niv.Values[7] := 0.0;
   Zulauf_AR_Niv.Values[8] := 0.0;
   Zulauf_AR_Niv.Values[9] := 0.0;
   Zulauf_AR_Niv.Values[10] := 0.0;
   Zulauf_AR_Niv.Values[11] := 0.0;
   Zulauf_AR_Niv.Values[12] := 0.0;
   Zulauf_AR_Niv.Values[13] := 0.0;
   Zulauf_AR_Niv.Values[14] := 0.0;
   Zulauf_AR_Niv.Values[15] := 0.0;
   Zulauf_AR_Niv.Values[16] := 0.0;
   Zulauf_AR_Niv.Values[17] := 0.0;
   Zulauf_AR_Niv.Values[18] := 0.0;
   Zulauf_AR_Niv.Values[19] := 0.0;
   Zulauf_AR_Niv.Values[20] := 0.0;
   Zulauf_AR_Niv.Values[21] := 0.0;
   Zulauf_AR_Niv.Values[22] := 0.0;
   Zulauf_AR_Niv.Values[23] := 0.0;
   Zulauf_AR_Niv.Values[24] := 0.0;
   Zulauf_AR_Niv.Values[25] := 0.0;
   Zulauf_AR_Niv.Values[26] := 0.0;
   Zulauf_AR_Niv.Values[27] := 0.0;
   Zulauf_AR_Niv.Values[28] := 0.0;
   Zulauf_AR_Niv.Values[29] := 0.0;
   Zulauf_AR_Niv.Values[30] := 0.0;
   Zulauf_AR_Niv.Values[31] := 0.0;
   Zulauf_AR_Niv.Values[32] := 0.0;
   Zulauf_AR_Niv.Values[33] := 0.0;
   Zulauf_AR_Niv.Values[34] := 0.0;
   Zulauf_AR_Niv.Values[35] := 0.0;
   Zulauf_AR_Niv.Values[36] := 0.0;
   Zulauf_AR_Niv.Values[37] := 0.0;
   Zulauf_AR_Niv.Values[38] := 0.0;
   Zulauf_AR_Niv.Values[39] := 0.0;
   Zulauf_AR_Niv.Values[40] := 0.0;
   Zulauf_AR_Niv.Values[41] := 0.0;
   Zulauf_AR_Niv.Values[42] := 0.0;
   Zulauf_AR_Niv.Values[43] := 0.0;
   Zulauf_AR_Niv.Values[44] := 0.0;
   Zulauf_AR_Niv.Values[45] := 0.0;
   Zulauf_AR_Niv.Values[46] := 0.0;
   Zulauf_AR_Niv.Values[47] := 0.0;
   Zulauf_AR_Niv.Values[48] := 0.0;
   Zulauf_AR_Niv.Values[49] := 0.0;
   Zulauf_AR_Niv.Values[50] := 0.0;
   Zulauf_AR_Niv.Values[51] := 0.0;
   Zulauf_AR_Niv.Values[52] := 0.0;
   Zulauf_AR_Niv.Values[53] := 0.0;
   Zulauf_AR_Niv.Values[54] := 0.0;
   Zulauf_AR_Niv.Values[55] := 0.0;
   Zulauf_AR_Niv.Values[56] := 0.0;
   Zulauf_AR_Niv.Values[57] := 0.0;
   Zulauf_AR_Niv.Values[58] := 0.0;
   Zulauf_AR_Niv.Values[59] := 0.0;
   Zulauf_AR_Niv.Values[60] := 0.0;
   Zulauf_AR_Niv.Values[61] := 0.0;
   Zulauf_AR_Niv.Values[62] := 0.0;
   Zulauf_AR_Niv.Values[63] := 0.0;
   Zulauf_AR_Niv.Values[64] := 0.0;
   Zulauf_AR_Niv.Values[65] := 0.0;
   Zulauf_AR_Niv.Values[66] := 0.0;
   Zulauf_AR_Niv.Values[67] := 0.0;
   Zulauf_AR_Niv.Values[68] := 0.0;
   Zulauf_AR_Niv.Values[69] := 0.0;
   Zulauf_AR_Niv.Values[70] := 0.0;
   Zulauf_AR_Niv.Values[71] := 0.0;
   Zulauf_AR_Niv.Values[72] := 0.0;
   Zulauf_AR_Niv.Values[73] := 0.0;
   Zulauf_AR_Niv.Values[74] := 0.0;
   Zulauf_AR_Niv.Values[75] := 0.0;
   Zulauf_AR_Niv.Values[76] := 0.0;
   Zulauf_AR_Niv.Values[77] := 0.0;
   Zulauf_AR_Niv.Values[78] := 0.0;
   Zulauf_AR_Niv.Values[79] := 0.0;
   Zulauf_AR_Niv.Values[80] := 0.0;
   Zulauf_AR_Niv.Values[81] := 0.0;
   Zulauf_AR_Niv.Values[82] := 0.0;
   Zulauf_AR_Niv.Values[83] := 0.0;
   Zulauf_AR_Niv.Values[84] := 0.0;
   Zulauf_AR_Niv.Values[85] := 0.0;
   Zulauf_AR_Niv.Values[86] := 0.0;
   Zulauf_AR_Niv.Values[87] := 0.0;
   Zulauf_AR_Niv.Values[88] := 0.0;
   Zulauf_AR_Niv.Values[89] := 0.0;
   Zulauf_AR_Niv.Values[90] := 0.0;
   Zulauf_AR_Niv.Values[91] := 0.0;
   Zulauf_AR_Niv.Values[92] := 0.0;
   Zulauf_AR_Niv.Values[93] := 0.0;
   Zulauf_AR_Niv.Values[94] := 0.0;
   Zulauf_AR_Niv.Values[95] := 0.0;
   Zulauf_AR_Niv.Values[96] := 0.0;
   Zulauf_AR_Niv.Values[97] := 0.0;
   Zulauf_AR_Niv.Values[98] := 0.0;
   Zulauf_AR_Niv.Values[99] := 0.0;
   Zulauf_AR_Niv.Values[100] := 0.0;
   Zulauf_AR_Niv.Values[101] := 0.0;
   Zulauf_AR_Niv.Values[102] := 0.0;
   Zulauf_AR_Niv.Values[103] := 0.0;
   Zulauf_AR_Niv.Values[104] := 0.0;
   Zulauf_AR_Niv.Values[105] := 0.0;
   Zulauf_AR_Niv.Values[106] := 0.0;
   Zulauf_AR_Niv.Values[107] := 0.0;
   Zulauf_AR_Niv.Values[108] := 0.0;
   Zulauf_AR_Niv.Values[109] := 0.0;
   Zulauf_AR_Niv.Values[110] := 0.0;
   Zulauf_AR_Niv.Values[111] := 0.0;
   Zulauf_AR_Niv.Values[112] := 0.0;
   Zulauf_AR_Niv.Values[113] := 0.0;
   Zulauf_AR_Niv.Values[114] := 0.0;
   Zulauf_AR_Niv.Values[115] := 0.0;
   Zulauf_AR_Niv.Values[116] := 0.0;
   Zulauf_AR_Niv.Values[117] := 0.0;
   Zulauf_AR_Niv.Values[118] := 0.0;
   Zulauf_AR_Niv.Values[119] := 0.0;
   Zulauf_AR_Temp.Values[0] := 0.0;
   Zulauf_AR_Temp.Values[1] := 0.0;
   Zulauf_AR_Temp.Values[2] := 0.0;
   Zulauf_AR_Temp.Values[3] := -0.2237052;
   Zulauf_AR_Temp.Values[4] := -0.2237052;
   Zulauf_AR_Temp.Values[5] := -0.2237052;
   Zulauf_AR_Temp.Values[6] := -0.2237052;
   Zulauf_AR_Temp.Values[7] := 1.867404;
   Zulauf_AR_Temp.Values[8] := 1.993996;
   Zulauf_AR_Temp.Values[9] := 1.908818;
   Zulauf_AR_Temp.Values[10] := 0.0;
   Zulauf_AR_Temp.Values[11] := 0.0;
   Zulauf_AR_Temp.Values[12] := 0.0;
   Zulauf_AR_Temp.Values[13] := 0.0;
   Zulauf_AR_Temp.Values[14] := 0.0;
   Zulauf_AR_Temp.Values[15] := 0.0;
   Zulauf_AR_Temp.Values[16] := 0.0;
   Zulauf_AR_Temp.Values[17] := 0.0;
   Zulauf_AR_Temp.Values[18] := 0.0;
   Zulauf_AR_Temp.Values[19] := 0.0;
   Zulauf_AR_Temp.Values[20] := 0.0;
   Zulauf_AR_Temp.Values[21] := 0.0;
   Zulauf_AR_Temp.Values[22] := 0.0;
   Zulauf_AR_Temp.Values[23] := 0.0;
   Zulauf_AR_Temp.Values[24] := 0.0;
   Zulauf_AR_Temp.Values[25] := 0.0;
   Zulauf_AR_Temp.Values[26] := 0.0;
   Zulauf_AR_Temp.Values[27] := 0.0;
   Zulauf_AR_Temp.Values[28] := 0.0;
   Zulauf_AR_Temp.Values[29] := 0.0;
   Zulauf_AR_Temp.Values[30] := 0.0;
   Zulauf_AR_Temp.Values[31] := 0.0;
   Zulauf_AR_Temp.Values[32] := 0.0;
   Zulauf_AR_Temp.Values[33] := 0.0;
   Zulauf_AR_Temp.Values[34] := 0.0;
   Zulauf_AR_Temp.Values[35] := 0.0;
   Zulauf_AR_Temp.Values[36] := 0.0;
   Zulauf_AR_Temp.Values[37] := 0.0;
   Zulauf_AR_Temp.Values[38] := 0.0;
   Zulauf_AR_Temp.Values[39] := 0.0;
   Zulauf_AR_Temp.Values[40] := 0.0;
   Zulauf_AR_Temp.Values[41] := 0.0;
   Zulauf_AR_Temp.Values[42] := 0.0;
   Zulauf_AR_Temp.Values[43] := 0.0;
   Zulauf_AR_Temp.Values[44] := 0.0;
   Zulauf_AR_Temp.Values[45] := 0.0;
   Zulauf_AR_Temp.Values[46] := 0.0;
   Zulauf_AR_Temp.Values[47] := 0.0;
   Zulauf_AR_Temp.Values[48] := 0.0;
   Zulauf_AR_Temp.Values[49] := 0.0;
   Zulauf_AR_Temp.Values[50] := 0.0;
   Zulauf_AR_Temp.Values[51] := 0.0;
   Zulauf_AR_Temp.Values[52] := 0.0;
   Zulauf_AR_Temp.Values[53] := 0.0;
   Zulauf_AR_Temp.Values[54] := 0.0;
   Zulauf_AR_Temp.Values[55] := 0.0;
   Zulauf_AR_Temp.Values[56] := 0.0;
   Zulauf_AR_Temp.Values[57] := 0.0;
   Zulauf_AR_Temp.Values[58] := 0.0;
   Zulauf_AR_Temp.Values[59] := 0.0;
   Zulauf_AR_Temp.Values[60] := 0.0;
   Zulauf_AR_Temp.Values[61] := 0.0;
   Zulauf_AR_Temp.Values[62] := 0.0;
   Zulauf_AR_Temp.Values[63] := 0.0;
   Zulauf_AR_Temp.Values[64] := 0.0;
   Zulauf_AR_Temp.Values[65] := 0.0;
   Zulauf_AR_Temp.Values[66] := 0.0;
   Zulauf_AR_Temp.Values[67] := 0.0;
   Zulauf_AR_Temp.Values[68] := 0.0;
   Zulauf_AR_Temp.Values[69] := 0.0;
   Zulauf_AR_Temp.Values[70] := 0.0;
   Zulauf_AR_Temp.Values[71] := 0.0;
   Zulauf_AR_Temp.Values[72] := 0.0;
   Zulauf_AR_Temp.Values[73] := 0.0;
   Zulauf_AR_Temp.Values[74] := 0.0;
   Zulauf_AR_Temp.Values[75] := 0.0;
   Zulauf_AR_Temp.Values[76] := 0.0;
   Zulauf_AR_Temp.Values[77] := 0.0;
   Zulauf_AR_Temp.Values[78] := 0.0;
   Zulauf_AR_Temp.Values[79] := 0.0;
   Zulauf_AR_Temp.Values[80] := 0.0;
   Zulauf_AR_Temp.Values[81] := 0.0;
   Zulauf_AR_Temp.Values[82] := 0.0;
   Zulauf_AR_Temp.Values[83] := 0.0;
   Zulauf_AR_Temp.Values[84] := 0.0;
   Zulauf_AR_Temp.Values[85] := 0.0;
   Zulauf_AR_Temp.Values[86] := 0.0;
   Zulauf_AR_Temp.Values[87] := 0.0;
   Zulauf_AR_Temp.Values[88] := 0.0;
   Zulauf_AR_Temp.Values[89] := 0.0;
   Zulauf_AR_Temp.Values[90] := 0.0;
   Zulauf_AR_Temp.Values[91] := 0.0;
   Zulauf_AR_Temp.Values[92] := 0.0;
   Zulauf_AR_Temp.Values[93] := 0.0;
   Zulauf_AR_Temp.Values[94] := 0.0;
   Zulauf_AR_Temp.Values[95] := 0.0;
   Zulauf_AR_Temp.Values[96] := 0.0;
   Zulauf_AR_Temp.Values[97] := 0.0;
   Zulauf_AR_Temp.Values[98] := 0.0;
   Zulauf_AR_Temp.Values[99] := 0.0;
   Zulauf_AR_Temp.Values[100] := 0.0;
   Zulauf_AR_Temp.Values[101] := 0.0;
   Zulauf_AR_Temp.Values[102] := 0.0;
   Zulauf_AR_Temp.Values[103] := 0.0;
   Zulauf_AR_Temp.Values[104] := 0.0;
   Zulauf_AR_Temp.Values[105] := 0.0;
   Zulauf_AR_Temp.Values[106] := 0.0;
   Zulauf_AR_Temp.Values[107] := 0.0;
   Zulauf_AR_Temp.Values[108] := 0.0;
   Zulauf_AR_Temp.Values[109] := 0.0;
   Zulauf_AR_Temp.Values[110] := 0.0;
   Zulauf_AR_Temp.Values[111] := 0.0;
   Zulauf_AR_Temp.Values[112] := 0.0;
   Zulauf_AR_Temp.Values[113] := 0.0;
   Zulauf_AR_Temp.Values[114] := 0.0;
   Zulauf_AR_Temp.Values[115] := 0.0;
   Zulauf_AR_Temp.Values[116] := 0.0;
   Zulauf_AR_Temp.Values[117] := 0.0;
   Zulauf_AR_Temp.Values[118] := 0.0;
   Zulauf_AR_Temp.Values[119] := 0.0;
   Zulauf_AR_DF.Values[0] := 4.441431;
   Zulauf_AR_DF.Values[1] := 4.441431;
   Zulauf_AR_DF.Values[2] := 4.441431;
   Zulauf_AR_DF.Values[3] := 58.8;
   Zulauf_AR_DF.Values[4] := 58.8;
   Zulauf_AR_DF.Values[5] := 58.8;
   Zulauf_AR_DF.Values[6] := 0.0;
   Zulauf_AR_DF.Values[7] := 0.0;
   Zulauf_AR_DF.Values[8] := 0.0;
   Zulauf_AR_DF.Values[9] := 0.0;
   Zulauf_AR_DF.Values[10] := 0.0;
   Zulauf_AR_DF.Values[11] := 0.0;
   Zulauf_AR_DF.Values[12] := 0.0;
   Zulauf_AR_DF.Values[13] := 0.0;
   Zulauf_AR_DF.Values[14] := 0.0;
   Zulauf_AR_DF.Values[15] := 0.0;
   Zulauf_AR_DF.Values[16] := 0.0;
   Zulauf_AR_DF.Values[17] := 0.0;
   Zulauf_AR_DF.Values[18] := 0.0;
   Zulauf_AR_DF.Values[19] := 0.0;
   Zulauf_AR_DF.Values[20] := 0.0;
   Zulauf_AR_DF.Values[21] := 0.0;
   Zulauf_AR_DF.Values[22] := 0.0;
   Zulauf_AR_DF.Values[23] := 0.0;
   Zulauf_AR_DF.Values[24] := 0.0;
   Zulauf_AR_DF.Values[25] := 0.0;
   Zulauf_AR_DF.Values[26] := 0.0;
   Zulauf_AR_DF.Values[27] := 0.0;
   Zulauf_AR_DF.Values[28] := 0.0;
   Zulauf_AR_DF.Values[29] := 0.0;
   Zulauf_AR_DF.Values[30] := 0.0;
   Zulauf_AR_DF.Values[31] := 0.0;
   Zulauf_AR_DF.Values[32] := 0.0;
   Zulauf_AR_DF.Values[33] := 0.0;
   Zulauf_AR_DF.Values[34] := 0.0;
   Zulauf_AR_DF.Values[35] := 0.0;
   Zulauf_AR_DF.Values[36] := 0.0;
   Zulauf_AR_DF.Values[37] := 0.0;
   Zulauf_AR_DF.Values[38] := 0.0;
   Zulauf_AR_DF.Values[39] := 0.0;
   Zulauf_AR_DF.Values[40] := 0.0;
   Zulauf_AR_DF.Values[41] := 0.0;
   Zulauf_AR_DF.Values[42] := 0.0;
   Zulauf_AR_DF.Values[43] := 0.0;
   Zulauf_AR_DF.Values[44] := 0.0;
   Zulauf_AR_DF.Values[45] := 0.0;
   Zulauf_AR_DF.Values[46] := 0.0;
   Zulauf_AR_DF.Values[47] := 0.0;
   Zulauf_AR_DF.Values[48] := 0.0;
   Zulauf_AR_DF.Values[49] := 0.0;
   Zulauf_AR_DF.Values[50] := 0.0;
   Zulauf_AR_DF.Values[51] := 0.0;
   Zulauf_AR_DF.Values[52] := 0.0;
   Zulauf_AR_DF.Values[53] := 0.0;
   Zulauf_AR_DF.Values[54] := 0.0;
   Zulauf_AR_DF.Values[55] := 0.0;
   Zulauf_AR_DF.Values[56] := 0.0;
   Zulauf_AR_DF.Values[57] := 0.0;
   Zulauf_AR_DF.Values[58] := 0.0;
   Zulauf_AR_DF.Values[59] := 0.0;
   Zulauf_AR_DF.Values[60] := 0.0;
   Zulauf_AR_DF.Values[61] := 0.0;
   Zulauf_AR_DF.Values[62] := 0.0;
   Zulauf_AR_DF.Values[63] := 0.0;
   Zulauf_AR_DF.Values[64] := 0.0;
   Zulauf_AR_DF.Values[65] := 0.0;
   Zulauf_AR_DF.Values[66] := 0.0;
   Zulauf_AR_DF.Values[67] := 0.0;
   Zulauf_AR_DF.Values[68] := 0.0;
   Zulauf_AR_DF.Values[69] := 0.0;
   Zulauf_AR_DF.Values[70] := 0.0;
   Zulauf_AR_DF.Values[71] := 0.0;
   Zulauf_AR_DF.Values[72] := 0.0;
   Zulauf_AR_DF.Values[73] := 0.0;
   Zulauf_AR_DF.Values[74] := 0.0;
   Zulauf_AR_DF.Values[75] := 0.0;
   Zulauf_AR_DF.Values[76] := 0.0;
   Zulauf_AR_DF.Values[77] := 0.0;
   Zulauf_AR_DF.Values[78] := 0.0;
   Zulauf_AR_DF.Values[79] := 0.0;
   Zulauf_AR_DF.Values[80] := 0.0;
   Zulauf_AR_DF.Values[81] := 0.0;
   Zulauf_AR_DF.Values[82] := 0.0;
   Zulauf_AR_DF.Values[83] := 0.0;
   Zulauf_AR_DF.Values[84] := 0.0;
   Zulauf_AR_DF.Values[85] := 0.0;
   Zulauf_AR_DF.Values[86] := 0.0;
   Zulauf_AR_DF.Values[87] := 0.0;
   Zulauf_AR_DF.Values[88] := 0.0;
   Zulauf_AR_DF.Values[89] := 0.0;
   Zulauf_AR_DF.Values[90] := 0.0;
   Zulauf_AR_DF.Values[91] := 0.0;
   Zulauf_AR_DF.Values[92] := 0.0;
   Zulauf_AR_DF.Values[93] := 0.0;
   Zulauf_AR_DF.Values[94] := 0.0;
   Zulauf_AR_DF.Values[95] := 0.0;
   Zulauf_AR_DF.Values[96] := 0.0;
   Zulauf_AR_DF.Values[97] := 0.0;
   Zulauf_AR_DF.Values[98] := 0.0;
   Zulauf_AR_DF.Values[99] := 0.0;
   Zulauf_AR_DF.Values[100] := 0.0;
   Zulauf_AR_DF.Values[101] := 0.0;
   Zulauf_AR_DF.Values[102] := 0.0;
   Zulauf_AR_DF.Values[103] := 0.0;
   Zulauf_AR_DF.Values[104] := 0.0;
   Zulauf_AR_DF.Values[105] := 0.0;
   Zulauf_AR_DF.Values[106] := 0.0;
   Zulauf_AR_DF.Values[107] := 0.0;
   Zulauf_AR_DF.Values[108] := 0.0;
   Zulauf_AR_DF.Values[109] := 0.0;
   Zulauf_AR_DF.Values[110] := 0.0;
   Zulauf_AR_DF.Values[111] := 0.0;
   Zulauf_AR_DF.Values[112] := 0.0;
   Zulauf_AR_DF.Values[113] := 0.0;
   Zulauf_AR_DF.Values[114] := 0.0;
   Zulauf_AR_DF.Values[115] := 0.0;
   Zulauf_AR_DF.Values[116] := 0.0;
   Zulauf_AR_DF.Values[117] := 0.0;
   Zulauf_AR_DF.Values[118] := 0.0;
   Zulauf_AR_DF.Values[119] := 0.0;
   BB1_AS1_SS.Values[0] := 0.0;
   BB1_AS1_SS.Values[1] := 0.0;
   BB1_AS1_SS.Values[2] := 0.0;
   BB1_AS1_SS.Values[3] := 0.0;
   BB1_AS1_SS.Values[4] := 0.0;
   BB1_AS1_SS.Values[5] := 0.0;
   BB1_AS1_SS.Values[6] := 0.0;
   BB1_AS1_SS.Values[7] := 0.0;
   BB1_AS1_SS.Values[8] := 0.0;
   BB1_AS1_SS.Values[9] := 0.0;
   BB1_AS1_SS.Values[10] := 0.0;
   BB1_AS1_SS.Values[11] := 0.0;
   BB1_AS1_SS.Values[12] := 0.0;
   BB1_AS1_SS.Values[13] := 0.0;
   BB1_AS1_SS.Values[14] := 0.0;
   BB1_AS1_SS.Values[15] := 0.0;
   BB1_AS1_SS.Values[16] := 0.0;
   BB1_AS1_SS.Values[17] := 0.0;
   BB1_AS1_SS.Values[18] := 0.0;
   BB1_AS1_SS.Values[19] := 0.0;
   BB1_AS1_SS.Values[20] := 0.0;
   BB1_AS1_SS.Values[21] := 0.0;
   BB1_AS1_SS.Values[22] := 0.0;
   BB1_AS1_SS.Values[23] := 0.0;
   BB1_AS1_SS.Values[24] := 0.0;
   BB1_AS1_SS.Values[25] := 0.0;
   BB1_AS1_SS.Values[26] := 0.0;
   BB1_AS1_SS.Values[27] := 0.0;
   BB1_AS1_SS.Values[28] := 0.0;
   BB1_AS1_SS.Values[29] := 0.0;
   BB1_AS1_SS.Values[30] := 0.0;
   BB1_AS1_SS.Values[31] := 0.0;
   BB1_AS1_SS.Values[32] := 0.0;
   BB1_AS1_SS.Values[33] := 0.0;
   BB1_AS1_SS.Values[34] := 0.0;
   BB1_AS1_SS.Values[35] := 0.0;
   BB1_AS1_SS.Values[36] := 0.0;
   BB1_AS1_SS.Values[37] := 0.0;
   BB1_AS1_SS.Values[38] := 0.0;
   BB1_AS1_SS.Values[39] := 0.0;
   BB1_AS1_SS.Values[40] := 0.0;
   BB1_AS1_SS.Values[41] := 0.0;
   BB1_AS1_SS.Values[42] := 0.0;
   BB1_AS1_SS.Values[43] := 0.0;
   BB1_AS1_SS.Values[44] := 0.0;
   BB1_AS1_SS.Values[45] := 0.0;
   BB1_AS1_SS.Values[46] := 0.0;
   BB1_AS1_SS.Values[47] := 0.0;
   BB1_AS1_SS.Values[48] := 0.0;
   BB1_AS1_SS.Values[49] := 0.0;
   BB1_AS1_SS.Values[50] := 0.0;
   BB1_AS1_SS.Values[51] := 0.0;
   BB1_AS1_SS.Values[52] := 0.0;
   BB1_AS1_SS.Values[53] := 0.0;
   BB1_AS1_SS.Values[54] := 0.0;
   BB1_AS1_SS.Values[55] := 0.0;
   BB1_AS1_SS.Values[56] := 0.0;
   BB1_AS1_SS.Values[57] := 0.0;
   BB1_AS1_SS.Values[58] := 0.0;
   BB1_AS1_SS.Values[59] := 0.0;
   BB1_AS1_SS.Values[60] := 0.0;
   BB1_AS1_SS.Values[61] := 0.0;
   BB1_AS1_SS.Values[62] := 0.0;
   BB1_AS1_SS.Values[63] := 0.0;
   BB1_AS1_SS.Values[64] := 0.0;
   BB1_AS1_SS.Values[65] := 0.0;
   BB1_AS1_SS.Values[66] := 0.0;
   BB1_AS1_SS.Values[67] := 0.0;
   BB1_AS1_SS.Values[68] := 0.0;
   BB1_AS1_SS.Values[69] := 0.0;
   BB1_AS1_SS.Values[70] := 0.0;
   BB1_AS1_SS.Values[71] := 0.0;
   BB1_AS1_SS.Values[72] := 0.0;
   BB1_AS1_SS.Values[73] := 0.0;
   BB1_AS1_SS.Values[74] := 0.0;
   BB1_AS1_SS.Values[75] := 0.0;
   BB1_AS1_SS.Values[76] := 0.0;
   BB1_AS1_SS.Values[77] := 0.0;
   BB1_AS1_SS.Values[78] := 0.0;
   BB1_AS1_SS.Values[79] := 0.0;
   BB1_AS1_SS.Values[80] := 0.0;
   BB1_AS1_SS.Values[81] := 0.0;
   BB1_AS1_SS.Values[82] := 0.0;
   BB1_AS1_SS.Values[83] := 0.0;
   BB1_AS1_SS.Values[84] := 0.0;
   BB1_AS1_SS.Values[85] := 0.0;
   BB1_AS1_SS.Values[86] := 0.0;
   BB1_AS1_SS.Values[87] := 0.0;
   BB1_AS1_SS.Values[88] := 0.0;
   BB1_AS1_SS.Values[89] := 0.0;
   BB1_AS1_SS.Values[90] := 0.0;
   BB1_AS1_SS.Values[91] := 0.0;
   BB1_AS1_SS.Values[92] := 0.0;
   BB1_AS1_SS.Values[93] := 0.0;
   BB1_AS1_SS.Values[94] := 0.0;
   BB1_AS1_SS.Values[95] := 0.0;
   BB1_AS1_SS.Values[96] := 0.0;
   BB1_AS1_SS.Values[97] := 0.0;
   BB1_AS1_SS.Values[98] := 0.0;
   BB1_AS1_SS.Values[99] := 0.0;
   BB1_AS1_SS.Values[100] := 0.0;
   BB1_AS1_SS.Values[101] := 0.0;
   BB1_AS1_SS.Values[102] := 0.0;
   BB1_AS1_SS.Values[103] := 0.0;
   BB1_AS1_SS.Values[104] := 0.0;
   BB1_AS1_SS.Values[105] := 0.0;
   BB1_AS1_SS.Values[106] := 0.0;
   BB1_AS1_SS.Values[107] := 0.0;
   BB1_AS1_SS.Values[108] := 0.0;
   BB1_AS1_SS.Values[109] := 0.0;
   BB1_AS1_SS.Values[110] := 0.0;
   BB1_AS1_SS.Values[111] := 0.0;
   BB1_AS1_SS.Values[112] := 0.0;
   BB1_AS1_SS.Values[113] := 0.0;
   BB1_AS1_SS.Values[114] := 0.0;
   BB1_AS1_SS.Values[115] := 0.0;
   BB1_AS1_SS.Values[116] := 0.0;
   BB1_AS1_SS.Values[117] := 0.0;
   BB1_AS1_SS.Values[118] := 0.0;
   BB1_AS1_SS.Values[119] := 0.0;
   BB1_AS2_SS.Values[0] := 12.64072;
   BB1_AS2_SS.Values[1] := 12.64072;
   BB1_AS2_SS.Values[2] := 12.64072;
   BB1_AS2_SS.Values[3] := 12.6362;
   BB1_AS2_SS.Values[4] := 12.64072;
   BB1_AS2_SS.Values[5] := 12.64072;
   BB1_AS2_SS.Values[6] := 12.64072;
   BB1_AS2_SS.Values[7] := 12.64072;
   BB1_AS2_SS.Values[8] := 12.64072;
   BB1_AS2_SS.Values[9] := 12.64072;
   BB1_AS2_SS.Values[10] := 23.0;
   BB1_AS2_SS.Values[11] := 23.1;
   BB1_AS2_SS.Values[12] := 23.1;
   BB1_AS2_SS.Values[13] := 23.1;
   BB1_AS2_SS.Values[14] := 23.1;
   BB1_AS2_SS.Values[15] := 23.0;
   BB1_AS2_SS.Values[16] := 23.0;
   BB1_AS2_SS.Values[17] := 23.1;
   BB1_AS2_SS.Values[18] := 23.1;
   BB1_AS2_SS.Values[19] := 23.1;
   BB1_AS2_SS.Values[20] := 23.1;
   BB1_AS2_SS.Values[21] := 23.1;
   BB1_AS2_SS.Values[22] := 23.1;
   BB1_AS2_SS.Values[23] := 23.1;
   BB1_AS2_SS.Values[24] := 23.1;
   BB1_AS2_SS.Values[25] := 23.0;
   BB1_AS2_SS.Values[26] := 23.1;
   BB1_AS2_SS.Values[27] := 23.1;
   BB1_AS2_SS.Values[28] := 23.1;
   BB1_AS2_SS.Values[29] := 23.1;
   BB1_AS2_SS.Values[30] := 0.0;
   BB1_AS2_SS.Values[31] := 0.0;
   BB1_AS2_SS.Values[32] := 0.0;
   BB1_AS2_SS.Values[33] := 0.0;
   BB1_AS2_SS.Values[34] := 0.0;
   BB1_AS2_SS.Values[35] := 0.0;
   BB1_AS2_SS.Values[36] := 0.0;
   BB1_AS2_SS.Values[37] := 0.0;
   BB1_AS2_SS.Values[38] := 0.0;
   BB1_AS2_SS.Values[39] := 0.0;
   BB1_AS2_SS.Values[40] := 0.0;
   BB1_AS2_SS.Values[41] := 0.0;
   BB1_AS2_SS.Values[42] := 0.0;
   BB1_AS2_SS.Values[43] := 0.0;
   BB1_AS2_SS.Values[44] := 0.0;
   BB1_AS2_SS.Values[45] := 0.0;
   BB1_AS2_SS.Values[46] := 0.0;
   BB1_AS2_SS.Values[47] := 0.0;
   BB1_AS2_SS.Values[48] := 0.0;
   BB1_AS2_SS.Values[49] := 0.0;
   BB1_AS2_SS.Values[50] := 0.0;
   BB1_AS2_SS.Values[51] := 0.0;
   BB1_AS2_SS.Values[52] := 0.0;
   BB1_AS2_SS.Values[53] := 0.0;
   BB1_AS2_SS.Values[54] := 0.0;
   BB1_AS2_SS.Values[55] := 0.0;
   BB1_AS2_SS.Values[56] := 0.0;
   BB1_AS2_SS.Values[57] := 0.0;
   BB1_AS2_SS.Values[58] := 0.0;
   BB1_AS2_SS.Values[59] := 0.0;
   BB1_AS2_SS.Values[60] := 0.0;
   BB1_AS2_SS.Values[61] := 0.0;
   BB1_AS2_SS.Values[62] := 0.0;
   BB1_AS2_SS.Values[63] := 0.0;
   BB1_AS2_SS.Values[64] := 0.0;
   BB1_AS2_SS.Values[65] := 0.0;
   BB1_AS2_SS.Values[66] := 0.0;
   BB1_AS2_SS.Values[67] := 0.0;
   BB1_AS2_SS.Values[68] := 0.0;
   BB1_AS2_SS.Values[69] := 0.0;
   BB1_AS2_SS.Values[70] := 0.0;
   BB1_AS2_SS.Values[71] := 0.0;
   BB1_AS2_SS.Values[72] := 0.0;
   BB1_AS2_SS.Values[73] := 0.0;
   BB1_AS2_SS.Values[74] := 0.0;
   BB1_AS2_SS.Values[75] := 0.0;
   BB1_AS2_SS.Values[76] := 0.0;
   BB1_AS2_SS.Values[77] := 0.0;
   BB1_AS2_SS.Values[78] := 0.0;
   BB1_AS2_SS.Values[79] := 0.0;
   BB1_AS2_SS.Values[80] := 0.0;
   BB1_AS2_SS.Values[81] := 0.0;
   BB1_AS2_SS.Values[82] := 0.0;
   BB1_AS2_SS.Values[83] := 0.0;
   BB1_AS2_SS.Values[84] := 0.0;
   BB1_AS2_SS.Values[85] := 0.0;
   BB1_AS2_SS.Values[86] := 0.0;
   BB1_AS2_SS.Values[87] := 0.0;
   BB1_AS2_SS.Values[88] := 0.0;
   BB1_AS2_SS.Values[89] := 0.0;
   BB1_AS2_SS.Values[90] := 0.0;
   BB1_AS2_SS.Values[91] := 0.0;
   BB1_AS2_SS.Values[92] := 0.0;
   BB1_AS2_SS.Values[93] := 0.0;
   BB1_AS2_SS.Values[94] := 0.0;
   BB1_AS2_SS.Values[95] := 0.0;
   BB1_AS2_SS.Values[96] := 0.0;
   BB1_AS2_SS.Values[97] := 0.0;
   BB1_AS2_SS.Values[98] := 0.0;
   BB1_AS2_SS.Values[99] := 0.0;
   BB1_AS2_SS.Values[100] := 0.0;
   BB1_AS2_SS.Values[101] := 0.0;
   BB1_AS2_SS.Values[102] := 0.0;
   BB1_AS2_SS.Values[103] := 0.0;
   BB1_AS2_SS.Values[104] := 0.0;
   BB1_AS2_SS.Values[105] := 0.0;
   BB1_AS2_SS.Values[106] := 0.0;
   BB1_AS2_SS.Values[107] := 0.0;
   BB1_AS2_SS.Values[108] := 0.0;
   BB1_AS2_SS.Values[109] := 0.0;
   BB1_AS2_SS.Values[110] := 0.0;
   BB1_AS2_SS.Values[111] := 0.0;
   BB1_AS2_SS.Values[112] := 0.0;
   BB1_AS2_SS.Values[113] := 0.0;
   BB1_AS2_SS.Values[114] := 0.0;
   BB1_AS2_SS.Values[115] := 0.0;
   BB1_AS2_SS.Values[116] := 0.0;
   BB1_AS2_SS.Values[117] := 0.0;
   BB1_AS2_SS.Values[118] := 0.0;
   BB1_AS2_SS.Values[119] := 0.0;
   BB2_AS1_SS.Values[0] := 0.036168;
   BB2_AS1_SS.Values[1] := 0.036168;
   BB2_AS1_SS.Values[2] := 0.031647;
   BB2_AS1_SS.Values[3] := 0.040689;
   BB2_AS1_SS.Values[4] := 0.040689;
   BB2_AS1_SS.Values[5] := 0.040689;
   BB2_AS1_SS.Values[6] := 0.036168;
   BB2_AS1_SS.Values[7] := 0.036168;
   BB2_AS1_SS.Values[8] := 0.040689;
   BB2_AS1_SS.Values[9] := 0.040689;
   BB2_AS1_SS.Values[10] := 0.0;
   BB2_AS1_SS.Values[11] := 0.0;
   BB2_AS1_SS.Values[12] := 0.0;
   BB2_AS1_SS.Values[13] := 0.0;
   BB2_AS1_SS.Values[14] := 0.0;
   BB2_AS1_SS.Values[15] := 0.0;
   BB2_AS1_SS.Values[16] := 0.0;
   BB2_AS1_SS.Values[17] := 0.0;
   BB2_AS1_SS.Values[18] := 0.0;
   BB2_AS1_SS.Values[19] := 0.0;
   BB2_AS1_SS.Values[20] := 0.0;
   BB2_AS1_SS.Values[21] := 0.0;
   BB2_AS1_SS.Values[22] := 0.0;
   BB2_AS1_SS.Values[23] := 0.0;
   BB2_AS1_SS.Values[24] := 0.0;
   BB2_AS1_SS.Values[25] := 0.0;
   BB2_AS1_SS.Values[26] := 0.0;
   BB2_AS1_SS.Values[27] := 0.0;
   BB2_AS1_SS.Values[28] := 0.0;
   BB2_AS1_SS.Values[29] := 0.0;
   BB2_AS1_SS.Values[30] := 0.0;
   BB2_AS1_SS.Values[31] := 0.0;
   BB2_AS1_SS.Values[32] := 0.0;
   BB2_AS1_SS.Values[33] := 0.0;
   BB2_AS1_SS.Values[34] := 0.0;
   BB2_AS1_SS.Values[35] := 0.0;
   BB2_AS1_SS.Values[36] := 0.0;
   BB2_AS1_SS.Values[37] := 0.0;
   BB2_AS1_SS.Values[38] := 0.0;
   BB2_AS1_SS.Values[39] := 0.0;
   BB2_AS1_SS.Values[40] := 0.0;
   BB2_AS1_SS.Values[41] := 0.0;
   BB2_AS1_SS.Values[42] := 0.0;
   BB2_AS1_SS.Values[43] := 0.0;
   BB2_AS1_SS.Values[44] := 0.0;
   BB2_AS1_SS.Values[45] := 0.0;
   BB2_AS1_SS.Values[46] := 0.0;
   BB2_AS1_SS.Values[47] := 0.0;
   BB2_AS1_SS.Values[48] := 0.0;
   BB2_AS1_SS.Values[49] := 0.0;
   BB2_AS1_SS.Values[50] := 0.0;
   BB2_AS1_SS.Values[51] := 0.0;
   BB2_AS1_SS.Values[52] := 0.0;
   BB2_AS1_SS.Values[53] := 0.0;
   BB2_AS1_SS.Values[54] := 0.0;
   BB2_AS1_SS.Values[55] := 0.0;
   BB2_AS1_SS.Values[56] := 0.0;
   BB2_AS1_SS.Values[57] := 0.0;
   BB2_AS1_SS.Values[58] := 0.0;
   BB2_AS1_SS.Values[59] := 0.0;
   BB2_AS1_SS.Values[60] := 0.0;
   BB2_AS1_SS.Values[61] := 0.0;
   BB2_AS1_SS.Values[62] := 0.0;
   BB2_AS1_SS.Values[63] := 0.0;
   BB2_AS1_SS.Values[64] := 0.0;
   BB2_AS1_SS.Values[65] := 0.0;
   BB2_AS1_SS.Values[66] := 0.0;
   BB2_AS1_SS.Values[67] := 0.0;
   BB2_AS1_SS.Values[68] := 0.0;
   BB2_AS1_SS.Values[69] := 0.0;
   BB2_AS1_SS.Values[70] := 0.0;
   BB2_AS1_SS.Values[71] := 0.0;
   BB2_AS1_SS.Values[72] := 0.0;
   BB2_AS1_SS.Values[73] := 0.0;
   BB2_AS1_SS.Values[74] := 0.0;
   BB2_AS1_SS.Values[75] := 0.0;
   BB2_AS1_SS.Values[76] := 0.0;
   BB2_AS1_SS.Values[77] := 0.0;
   BB2_AS1_SS.Values[78] := 0.0;
   BB2_AS1_SS.Values[79] := 0.0;
   BB2_AS1_SS.Values[80] := 0.0;
   BB2_AS1_SS.Values[81] := 0.0;
   BB2_AS1_SS.Values[82] := 0.0;
   BB2_AS1_SS.Values[83] := 0.0;
   BB2_AS1_SS.Values[84] := 0.0;
   BB2_AS1_SS.Values[85] := 0.0;
   BB2_AS1_SS.Values[86] := 0.0;
   BB2_AS1_SS.Values[87] := 0.0;
   BB2_AS1_SS.Values[88] := 0.0;
   BB2_AS1_SS.Values[89] := 0.0;
   BB2_AS1_SS.Values[90] := 0.0;
   BB2_AS1_SS.Values[91] := 0.0;
   BB2_AS1_SS.Values[92] := 0.0;
   BB2_AS1_SS.Values[93] := 0.0;
   BB2_AS1_SS.Values[94] := 0.0;
   BB2_AS1_SS.Values[95] := 0.0;
   BB2_AS1_SS.Values[96] := 0.0;
   BB2_AS1_SS.Values[97] := 0.0;
   BB2_AS1_SS.Values[98] := 0.0;
   BB2_AS1_SS.Values[99] := 0.0;
   BB2_AS1_SS.Values[100] := 0.0;
   BB2_AS1_SS.Values[101] := 0.0;
   BB2_AS1_SS.Values[102] := 0.0;
   BB2_AS1_SS.Values[103] := 0.0;
   BB2_AS1_SS.Values[104] := 0.0;
   BB2_AS1_SS.Values[105] := 0.0;
   BB2_AS1_SS.Values[106] := 0.0;
   BB2_AS1_SS.Values[107] := 0.0;
   BB2_AS1_SS.Values[108] := 0.0;
   BB2_AS1_SS.Values[109] := 0.0;
   BB2_AS1_SS.Values[110] := 0.0;
   BB2_AS1_SS.Values[111] := 0.0;
   BB2_AS1_SS.Values[112] := 0.0;
   BB2_AS1_SS.Values[113] := 0.0;
   BB2_AS1_SS.Values[114] := 0.0;
   BB2_AS1_SS.Values[115] := 0.0;
   BB2_AS1_SS.Values[116] := 0.0;
   BB2_AS1_SS.Values[117] := 0.0;
   BB2_AS1_SS.Values[118] := 0.0;
   BB2_AS1_SS.Values[119] := 0.0;
   BB2_AS2_SS.Values[0] := 0.140151;
   BB2_AS2_SS.Values[1] := 0.140151;
   BB2_AS2_SS.Values[2] := 0.140151;
   BB2_AS2_SS.Values[3] := 0.140151;
   BB2_AS2_SS.Values[4] := 0.140151;
   BB2_AS2_SS.Values[5] := 0.140151;
   BB2_AS2_SS.Values[6] := 0.140151;
   BB2_AS2_SS.Values[7] := 0.140151;
   BB2_AS2_SS.Values[8] := 0.140151;
   BB2_AS2_SS.Values[9] := 0.140151;
   BB2_AS2_SS.Values[10] := 23.9;
   BB2_AS2_SS.Values[11] := 23.9;
   BB2_AS2_SS.Values[12] := 23.9;
   BB2_AS2_SS.Values[13] := 23.9;
   BB2_AS2_SS.Values[14] := 23.9;
   BB2_AS2_SS.Values[15] := 23.9;
   BB2_AS2_SS.Values[16] := 23.9;
   BB2_AS2_SS.Values[17] := 23.9;
   BB2_AS2_SS.Values[18] := 23.9;
   BB2_AS2_SS.Values[19] := 23.9;
   BB2_AS2_SS.Values[20] := 23.9;
   BB2_AS2_SS.Values[21] := 23.9;
   BB2_AS2_SS.Values[22] := 23.9;
   BB2_AS2_SS.Values[23] := 23.9;
   BB2_AS2_SS.Values[24] := 23.9;
   BB2_AS2_SS.Values[25] := 23.9;
   BB2_AS2_SS.Values[26] := 23.9;
   BB2_AS2_SS.Values[27] := 23.9;
   BB2_AS2_SS.Values[28] := 23.9;
   BB2_AS2_SS.Values[29] := 23.9;
   BB2_AS2_SS.Values[30] := 0.0;
   BB2_AS2_SS.Values[31] := 0.0;
   BB2_AS2_SS.Values[32] := 0.0;
   BB2_AS2_SS.Values[33] := 0.0;
   BB2_AS2_SS.Values[34] := 0.0;
   BB2_AS2_SS.Values[35] := 0.0;
   BB2_AS2_SS.Values[36] := 0.0;
   BB2_AS2_SS.Values[37] := 0.0;
   BB2_AS2_SS.Values[38] := 0.0;
   BB2_AS2_SS.Values[39] := 0.0;
   BB2_AS2_SS.Values[40] := 0.0;
   BB2_AS2_SS.Values[41] := 0.0;
   BB2_AS2_SS.Values[42] := 0.0;
   BB2_AS2_SS.Values[43] := 0.0;
   BB2_AS2_SS.Values[44] := 0.0;
   BB2_AS2_SS.Values[45] := 0.0;
   BB2_AS2_SS.Values[46] := 0.0;
   BB2_AS2_SS.Values[47] := 0.0;
   BB2_AS2_SS.Values[48] := 0.0;
   BB2_AS2_SS.Values[49] := 0.0;
   BB2_AS2_SS.Values[50] := 0.0;
   BB2_AS2_SS.Values[51] := 0.0;
   BB2_AS2_SS.Values[52] := 0.0;
   BB2_AS2_SS.Values[53] := 0.0;
   BB2_AS2_SS.Values[54] := 0.0;
   BB2_AS2_SS.Values[55] := 0.0;
   BB2_AS2_SS.Values[56] := 0.0;
   BB2_AS2_SS.Values[57] := 0.0;
   BB2_AS2_SS.Values[58] := 0.0;
   BB2_AS2_SS.Values[59] := 0.0;
   BB2_AS2_SS.Values[60] := 0.0;
   BB2_AS2_SS.Values[61] := 0.0;
   BB2_AS2_SS.Values[62] := 0.0;
   BB2_AS2_SS.Values[63] := 0.0;
   BB2_AS2_SS.Values[64] := 0.0;
   BB2_AS2_SS.Values[65] := 0.0;
   BB2_AS2_SS.Values[66] := 0.0;
   BB2_AS2_SS.Values[67] := 0.0;
   BB2_AS2_SS.Values[68] := 0.0;
   BB2_AS2_SS.Values[69] := 0.0;
   BB2_AS2_SS.Values[70] := 0.0;
   BB2_AS2_SS.Values[71] := 0.0;
   BB2_AS2_SS.Values[72] := 0.0;
   BB2_AS2_SS.Values[73] := 0.0;
   BB2_AS2_SS.Values[74] := 0.0;
   BB2_AS2_SS.Values[75] := 0.0;
   BB2_AS2_SS.Values[76] := 0.0;
   BB2_AS2_SS.Values[77] := 0.0;
   BB2_AS2_SS.Values[78] := 0.0;
   BB2_AS2_SS.Values[79] := 0.0;
   BB2_AS2_SS.Values[80] := 0.0;
   BB2_AS2_SS.Values[81] := 0.0;
   BB2_AS2_SS.Values[82] := 0.0;
   BB2_AS2_SS.Values[83] := 0.0;
   BB2_AS2_SS.Values[84] := 0.0;
   BB2_AS2_SS.Values[85] := 0.0;
   BB2_AS2_SS.Values[86] := 0.0;
   BB2_AS2_SS.Values[87] := 0.0;
   BB2_AS2_SS.Values[88] := 0.0;
   BB2_AS2_SS.Values[89] := 0.0;
   BB2_AS2_SS.Values[90] := 0.0;
   BB2_AS2_SS.Values[91] := 0.0;
   BB2_AS2_SS.Values[92] := 0.0;
   BB2_AS2_SS.Values[93] := 0.0;
   BB2_AS2_SS.Values[94] := 0.0;
   BB2_AS2_SS.Values[95] := 0.0;
   BB2_AS2_SS.Values[96] := 0.0;
   BB2_AS2_SS.Values[97] := 0.0;
   BB2_AS2_SS.Values[98] := 0.0;
   BB2_AS2_SS.Values[99] := 0.0;
   BB2_AS2_SS.Values[100] := 0.0;
   BB2_AS2_SS.Values[101] := 0.0;
   BB2_AS2_SS.Values[102] := 0.0;
   BB2_AS2_SS.Values[103] := 0.0;
   BB2_AS2_SS.Values[104] := 0.0;
   BB2_AS2_SS.Values[105] := 0.0;
   BB2_AS2_SS.Values[106] := 0.0;
   BB2_AS2_SS.Values[107] := 0.0;
   BB2_AS2_SS.Values[108] := 0.0;
   BB2_AS2_SS.Values[109] := 0.0;
   BB2_AS2_SS.Values[110] := 0.0;
   BB2_AS2_SS.Values[111] := 0.0;
   BB2_AS2_SS.Values[112] := 0.0;
   BB2_AS2_SS.Values[113] := 0.0;
   BB2_AS2_SS.Values[114] := 0.0;
   BB2_AS2_SS.Values[115] := 0.0;
   BB2_AS2_SS.Values[116] := 0.0;
   BB2_AS2_SS.Values[117] := 0.0;
   BB2_AS2_SS.Values[118] := 0.0;
   BB2_AS2_SS.Values[119] := 0.0;
   BB1_O2.Values[0] := 0.5212713;
   BB1_O2.Values[1] := 0.5212713;
   BB1_O2.Values[2] := 0.5212713;
   BB1_O2.Values[3] := 0.524436;
   BB1_O2.Values[4] := 0.524436;
   BB1_O2.Values[5] := 0.524436;
   BB1_O2.Values[6] := 0.524436;
   BB1_O2.Values[7] := 0.524436;
   BB1_O2.Values[8] := 0.528957;
   BB1_O2.Values[9] := 0.5294091;
   BB1_O2.Values[10] := 0.528957;
   BB1_O2.Values[11] := 0.528957;
   BB1_O2.Values[12] := 0.5294091;
   BB1_O2.Values[13] := 0.5352864;
   BB1_O2.Values[14] := 0.5357385;
   BB1_O2.Values[15] := 0.5357385;
   BB1_O2.Values[16] := 0.5352864;
   BB1_O2.Values[17] := 0.5352864;
   BB1_O2.Values[18] := 0.5352864;
   BB1_O2.Values[19] := 0.547041;
   BB1_O2.Values[20] := 0.547041;
   BB1_O2.Values[21] := 0.547041;
   BB1_O2.Values[22] := 0.547041;
   BB1_O2.Values[23] := 0.5465889;
   BB1_O2.Values[24] := 0.5578914;
   BB1_O2.Values[25] := 0.5578914;
   BB1_O2.Values[26] := 0.5578914;
   BB1_O2.Values[27] := 0.5212713;
   BB1_O2.Values[28] := 0.5212713;
   BB1_O2.Values[29] := 0.5212713;
   BB1_O2.Values[30] := 0.0;
   BB1_O2.Values[31] := 0.0;
   BB1_O2.Values[32] := 0.0;
   BB1_O2.Values[33] := 0.0;
   BB1_O2.Values[34] := 0.0;
   BB1_O2.Values[35] := 0.0;
   BB1_O2.Values[36] := 0.0;
   BB1_O2.Values[37] := 0.0;
   BB1_O2.Values[38] := 0.0;
   BB1_O2.Values[39] := 0.0;
   BB1_O2.Values[40] := 0.0;
   BB1_O2.Values[41] := 0.0;
   BB1_O2.Values[42] := 0.0;
   BB1_O2.Values[43] := 0.0;
   BB1_O2.Values[44] := 0.0;
   BB1_O2.Values[45] := 0.0;
   BB1_O2.Values[46] := 0.0;
   BB1_O2.Values[47] := 0.0;
   BB1_O2.Values[48] := 0.0;
   BB1_O2.Values[49] := 0.0;
   BB1_O2.Values[50] := 0.0;
   BB1_O2.Values[51] := 0.0;
   BB1_O2.Values[52] := 0.0;
   BB1_O2.Values[53] := 0.0;
   BB1_O2.Values[54] := 0.0;
   BB1_O2.Values[55] := 0.0;
   BB1_O2.Values[56] := 0.0;
   BB1_O2.Values[57] := 0.0;
   BB1_O2.Values[58] := 0.0;
   BB1_O2.Values[59] := 0.0;
   BB1_O2.Values[60] := 0.0;
   BB1_O2.Values[61] := 0.0;
   BB1_O2.Values[62] := 0.0;
   BB1_O2.Values[63] := 0.0;
   BB1_O2.Values[64] := 0.0;
   BB1_O2.Values[65] := 0.0;
   BB1_O2.Values[66] := 0.0;
   BB1_O2.Values[67] := 0.0;
   BB1_O2.Values[68] := 0.0;
   BB1_O2.Values[69] := 0.0;
   BB1_O2.Values[70] := 0.0;
   BB1_O2.Values[71] := 0.0;
   BB1_O2.Values[72] := 0.0;
   BB1_O2.Values[73] := 0.0;
   BB1_O2.Values[74] := 0.0;
   BB1_O2.Values[75] := 0.0;
   BB1_O2.Values[76] := 0.0;
   BB1_O2.Values[77] := 0.0;
   BB1_O2.Values[78] := 0.0;
   BB1_O2.Values[79] := 0.0;
   BB1_O2.Values[80] := 0.0;
   BB1_O2.Values[81] := 0.0;
   BB1_O2.Values[82] := 0.0;
   BB1_O2.Values[83] := 0.0;
   BB1_O2.Values[84] := 0.0;
   BB1_O2.Values[85] := 0.0;
   BB1_O2.Values[86] := 0.0;
   BB1_O2.Values[87] := 0.0;
   BB1_O2.Values[88] := 0.0;
   BB1_O2.Values[89] := 0.0;
   BB1_O2.Values[90] := 0.0;
   BB1_O2.Values[91] := 0.0;
   BB1_O2.Values[92] := 0.0;
   BB1_O2.Values[93] := 0.0;
   BB1_O2.Values[94] := 0.0;
   BB1_O2.Values[95] := 0.0;
   BB1_O2.Values[96] := 0.0;
   BB1_O2.Values[97] := 0.0;
   BB1_O2.Values[98] := 0.0;
   BB1_O2.Values[99] := 0.0;
   BB1_O2.Values[100] := 0.0;
   BB1_O2.Values[101] := 0.0;
   BB1_O2.Values[102] := 0.0;
   BB1_O2.Values[103] := 0.0;
   BB1_O2.Values[104] := 0.0;
   BB1_O2.Values[105] := 0.0;
   BB1_O2.Values[106] := 0.0;
   BB1_O2.Values[107] := 0.0;
   BB1_O2.Values[108] := 0.0;
   BB1_O2.Values[109] := 0.0;
   BB1_O2.Values[110] := 0.0;
   BB1_O2.Values[111] := 0.0;
   BB1_O2.Values[112] := 0.0;
   BB1_O2.Values[113] := 0.0;
   BB1_O2.Values[114] := 0.0;
   BB1_O2.Values[115] := 0.0;
   BB1_O2.Values[116] := 0.0;
   BB1_O2.Values[117] := 0.0;
   BB1_O2.Values[118] := 0.0;
   BB1_O2.Values[119] := 0.0;
   BB1_Temp.Values[0] := 14.53728;
   BB1_Temp.Values[1] := 14.53728;
   BB1_Temp.Values[2] := 14.53728;
   BB1_Temp.Values[3] := 14.53728;
   BB1_Temp.Values[4] := 14.53728;
   BB1_Temp.Values[5] := 14.53728;
   BB1_Temp.Values[6] := 14.53275;
   BB1_Temp.Values[7] := 14.53728;
   BB1_Temp.Values[8] := 14.53728;
   BB1_Temp.Values[9] := 14.53275;
   BB1_Temp.Values[10] := 14.53728;
   BB1_Temp.Values[11] := 14.53728;
   BB1_Temp.Values[12] := 14.53275;
   BB1_Temp.Values[13] := 14.53728;
   BB1_Temp.Values[14] := 14.53728;
   BB1_Temp.Values[15] := 14.53275;
   BB1_Temp.Values[16] := 14.53275;
   BB1_Temp.Values[17] := 14.53275;
   BB1_Temp.Values[18] := 14.53728;
   BB1_Temp.Values[19] := 14.53728;
   BB1_Temp.Values[20] := 14.53728;
   BB1_Temp.Values[21] := 14.53728;
   BB1_Temp.Values[22] := 14.53728;
   BB1_Temp.Values[23] := 14.53275;
   BB1_Temp.Values[24] := 14.53275;
   BB1_Temp.Values[25] := 14.53275;
   BB1_Temp.Values[26] := 14.53728;
   BB1_Temp.Values[27] := 14.53728;
   BB1_Temp.Values[28] := 14.53275;
   BB1_Temp.Values[29] := 14.53728;
   BB1_Temp.Values[30] := 0.0;
   BB1_Temp.Values[31] := 0.0;
   BB1_Temp.Values[32] := 0.0;
   BB1_Temp.Values[33] := 0.0;
   BB1_Temp.Values[34] := 0.0;
   BB1_Temp.Values[35] := 0.0;
   BB1_Temp.Values[36] := 0.0;
   BB1_Temp.Values[37] := 0.0;
   BB1_Temp.Values[38] := 0.0;
   BB1_Temp.Values[39] := 0.0;
   BB1_Temp.Values[40] := 0.0;
   BB1_Temp.Values[41] := 0.0;
   BB1_Temp.Values[42] := 0.0;
   BB1_Temp.Values[43] := 0.0;
   BB1_Temp.Values[44] := 0.0;
   BB1_Temp.Values[45] := 0.0;
   BB1_Temp.Values[46] := 0.0;
   BB1_Temp.Values[47] := 0.0;
   BB1_Temp.Values[48] := 0.0;
   BB1_Temp.Values[49] := 0.0;
   BB1_Temp.Values[50] := 0.0;
   BB1_Temp.Values[51] := 0.0;
   BB1_Temp.Values[52] := 0.0;
   BB1_Temp.Values[53] := 0.0;
   BB1_Temp.Values[54] := 0.0;
   BB1_Temp.Values[55] := 0.0;
   BB1_Temp.Values[56] := 0.0;
   BB1_Temp.Values[57] := 0.0;
   BB1_Temp.Values[58] := 0.0;
   BB1_Temp.Values[59] := 0.0;
   BB1_Temp.Values[60] := 0.0;
   BB1_Temp.Values[61] := 0.0;
   BB1_Temp.Values[62] := 0.0;
   BB1_Temp.Values[63] := 0.0;
   BB1_Temp.Values[64] := 0.0;
   BB1_Temp.Values[65] := 0.0;
   BB1_Temp.Values[66] := 0.0;
   BB1_Temp.Values[67] := 0.0;
   BB1_Temp.Values[68] := 0.0;
   BB1_Temp.Values[69] := 0.0;
   BB1_Temp.Values[70] := 0.0;
   BB1_Temp.Values[71] := 0.0;
   BB1_Temp.Values[72] := 0.0;
   BB1_Temp.Values[73] := 0.0;
   BB1_Temp.Values[74] := 0.0;
   BB1_Temp.Values[75] := 0.0;
   BB1_Temp.Values[76] := 0.0;
   BB1_Temp.Values[77] := 0.0;
   BB1_Temp.Values[78] := 0.0;
   BB1_Temp.Values[79] := 0.0;
   BB1_Temp.Values[80] := 0.0;
   BB1_Temp.Values[81] := 0.0;
   BB1_Temp.Values[82] := 0.0;
   BB1_Temp.Values[83] := 0.0;
   BB1_Temp.Values[84] := 0.0;
   BB1_Temp.Values[85] := 0.0;
   BB1_Temp.Values[86] := 0.0;
   BB1_Temp.Values[87] := 0.0;
   BB1_Temp.Values[88] := 0.0;
   BB1_Temp.Values[89] := 0.0;
   BB1_Temp.Values[90] := 0.0;
   BB1_Temp.Values[91] := 0.0;
   BB1_Temp.Values[92] := 0.0;
   BB1_Temp.Values[93] := 0.0;
   BB1_Temp.Values[94] := 0.0;
   BB1_Temp.Values[95] := 0.0;
   BB1_Temp.Values[96] := 0.0;
   BB1_Temp.Values[97] := 0.0;
   BB1_Temp.Values[98] := 0.0;
   BB1_Temp.Values[99] := 0.0;
   BB1_Temp.Values[100] := 0.0;
   BB1_Temp.Values[101] := 0.0;
   BB1_Temp.Values[102] := 0.0;
   BB1_Temp.Values[103] := 0.0;
   BB1_Temp.Values[104] := 0.0;
   BB1_Temp.Values[105] := 0.0;
   BB1_Temp.Values[106] := 0.0;
   BB1_Temp.Values[107] := 0.0;
   BB1_Temp.Values[108] := 0.0;
   BB1_Temp.Values[109] := 0.0;
   BB1_Temp.Values[110] := 0.0;
   BB1_Temp.Values[111] := 0.0;
   BB1_Temp.Values[112] := 0.0;
   BB1_Temp.Values[113] := 0.0;
   BB1_Temp.Values[114] := 0.0;
   BB1_Temp.Values[115] := 0.0;
   BB1_Temp.Values[116] := 0.0;
   BB1_Temp.Values[117] := 0.0;
   BB1_Temp.Values[118] := 0.0;
   BB1_Temp.Values[119] := 0.0;
   BB2_O2.Values[0] := 0.6198291;
   BB2_O2.Values[1] := 0.6198291;
   BB2_O2.Values[2] := 0.6202812;
   BB2_O2.Values[3] := 0.6257064;
   BB2_O2.Values[4] := 0.6257064;
   BB2_O2.Values[5] := 0.6257064;
   BB2_O2.Values[6] := 0.6257064;
   BB2_O2.Values[7] := 0.6257064;
   BB2_O2.Values[8] := 0.6311316;
   BB2_O2.Values[9] := 0.6306795;
   BB2_O2.Values[10] := 0.6311316;
   BB2_O2.Values[11] := 0.6306795;
   BB2_O2.Values[12] := 0.6306795;
   BB2_O2.Values[13] := 0.6352005;
   BB2_O2.Values[14] := 0.6356526;
   BB2_O2.Values[15] := 0.6356526;
   BB2_O2.Values[16] := 0.6356526;
   BB2_O2.Values[17] := 0.6356526;
   BB2_O2.Values[18] := 0.6356526;
   BB2_O2.Values[19] := 0.6388173;
   BB2_O2.Values[20] := 0.6383652;
   BB2_O2.Values[21] := 0.6388173;
   BB2_O2.Values[22] := 0.6388173;
   BB2_O2.Values[23] := 0.6388173;
   BB2_O2.Values[24] := 0.6415299;
   BB2_O2.Values[25] := 0.641982;
   BB2_O2.Values[26] := 0.6415299;
   BB2_O2.Values[27] := 0.6198291;
   BB2_O2.Values[28] := 0.6198291;
   BB2_O2.Values[29] := 0.6198291;
   BB2_O2.Values[30] := 0.0;
   BB2_O2.Values[31] := 0.0;
   BB2_O2.Values[32] := 0.0;
   BB2_O2.Values[33] := 0.0;
   BB2_O2.Values[34] := 0.0;
   BB2_O2.Values[35] := 0.0;
   BB2_O2.Values[36] := 0.0;
   BB2_O2.Values[37] := 0.0;
   BB2_O2.Values[38] := 0.0;
   BB2_O2.Values[39] := 0.0;
   BB2_O2.Values[40] := 0.0;
   BB2_O2.Values[41] := 0.0;
   BB2_O2.Values[42] := 0.0;
   BB2_O2.Values[43] := 0.0;
   BB2_O2.Values[44] := 0.0;
   BB2_O2.Values[45] := 0.0;
   BB2_O2.Values[46] := 0.0;
   BB2_O2.Values[47] := 0.0;
   BB2_O2.Values[48] := 0.0;
   BB2_O2.Values[49] := 0.0;
   BB2_O2.Values[50] := 0.0;
   BB2_O2.Values[51] := 0.0;
   BB2_O2.Values[52] := 0.0;
   BB2_O2.Values[53] := 0.0;
   BB2_O2.Values[54] := 0.0;
   BB2_O2.Values[55] := 0.0;
   BB2_O2.Values[56] := 0.0;
   BB2_O2.Values[57] := 0.0;
   BB2_O2.Values[58] := 0.0;
   BB2_O2.Values[59] := 0.0;
   BB2_O2.Values[60] := 0.0;
   BB2_O2.Values[61] := 0.0;
   BB2_O2.Values[62] := 0.0;
   BB2_O2.Values[63] := 0.0;
   BB2_O2.Values[64] := 0.0;
   BB2_O2.Values[65] := 0.0;
   BB2_O2.Values[66] := 0.0;
   BB2_O2.Values[67] := 0.0;
   BB2_O2.Values[68] := 0.0;
   BB2_O2.Values[69] := 0.0;
   BB2_O2.Values[70] := 0.0;
   BB2_O2.Values[71] := 0.0;
   BB2_O2.Values[72] := 0.0;
   BB2_O2.Values[73] := 0.0;
   BB2_O2.Values[74] := 0.0;
   BB2_O2.Values[75] := 0.0;
   BB2_O2.Values[76] := 0.0;
   BB2_O2.Values[77] := 0.0;
   BB2_O2.Values[78] := 0.0;
   BB2_O2.Values[79] := 0.0;
   BB2_O2.Values[80] := 0.0;
   BB2_O2.Values[81] := 0.0;
   BB2_O2.Values[82] := 0.0;
   BB2_O2.Values[83] := 0.0;
   BB2_O2.Values[84] := 0.0;
   BB2_O2.Values[85] := 0.0;
   BB2_O2.Values[86] := 0.0;
   BB2_O2.Values[87] := 0.0;
   BB2_O2.Values[88] := 0.0;
   BB2_O2.Values[89] := 0.0;
   BB2_O2.Values[90] := 0.0;
   BB2_O2.Values[91] := 0.0;
   BB2_O2.Values[92] := 0.0;
   BB2_O2.Values[93] := 0.0;
   BB2_O2.Values[94] := 0.0;
   BB2_O2.Values[95] := 0.0;
   BB2_O2.Values[96] := 0.0;
   BB2_O2.Values[97] := 0.0;
   BB2_O2.Values[98] := 0.0;
   BB2_O2.Values[99] := 0.0;
   BB2_O2.Values[100] := 0.0;
   BB2_O2.Values[101] := 0.0;
   BB2_O2.Values[102] := 0.0;
   BB2_O2.Values[103] := 0.0;
   BB2_O2.Values[104] := 0.0;
   BB2_O2.Values[105] := 0.0;
   BB2_O2.Values[106] := 0.0;
   BB2_O2.Values[107] := 0.0;
   BB2_O2.Values[108] := 0.0;
   BB2_O2.Values[109] := 0.0;
   BB2_O2.Values[110] := 0.0;
   BB2_O2.Values[111] := 0.0;
   BB2_O2.Values[112] := 0.0;
   BB2_O2.Values[113] := 0.0;
   BB2_O2.Values[114] := 0.0;
   BB2_O2.Values[115] := 0.0;
   BB2_O2.Values[116] := 0.0;
   BB2_O2.Values[117] := 0.0;
   BB2_O2.Values[118] := 0.0;
   BB2_O2.Values[119] := 0.0;
   BB2_Temp.Values[0] := 14.39034;
   BB2_Temp.Values[1] := 14.39034;
   BB2_Temp.Values[2] := 14.38808;
   BB2_Temp.Values[3] := 14.39034;
   BB2_Temp.Values[4] := 14.39034;
   BB2_Temp.Values[5] := 14.38808;
   BB2_Temp.Values[6] := 14.39034;
   BB2_Temp.Values[7] := 14.39034;
   BB2_Temp.Values[8] := 14.38356;
   BB2_Temp.Values[9] := 14.38356;
   BB2_Temp.Values[10] := 14.38356;
   BB2_Temp.Values[11] := 14.38356;
   BB2_Temp.Values[12] := 14.38582;
   BB2_Temp.Values[13] := 14.38582;
   BB2_Temp.Values[14] := 14.38356;
   BB2_Temp.Values[15] := 14.38356;
   BB2_Temp.Values[16] := 14.38582;
   BB2_Temp.Values[17] := 14.38582;
   BB2_Temp.Values[18] := 14.38582;
   BB2_Temp.Values[19] := 14.38808;
   BB2_Temp.Values[20] := 14.39034;
   BB2_Temp.Values[21] := 14.39034;
   BB2_Temp.Values[22] := 14.38808;
   BB2_Temp.Values[23] := 14.38808;
   BB2_Temp.Values[24] := 14.39034;
   BB2_Temp.Values[25] := 14.38808;
   BB2_Temp.Values[26] := 14.39034;
   BB2_Temp.Values[27] := 14.38808;
   BB2_Temp.Values[28] := 14.39034;
   BB2_Temp.Values[29] := 14.39034;
   BB2_Temp.Values[30] := 0.0;
   BB2_Temp.Values[31] := 0.0;
   BB2_Temp.Values[32] := 0.0;
   BB2_Temp.Values[33] := 0.0;
   BB2_Temp.Values[34] := 0.0;
   BB2_Temp.Values[35] := 0.0;
   BB2_Temp.Values[36] := 0.0;
   BB2_Temp.Values[37] := 0.0;
   BB2_Temp.Values[38] := 0.0;
   BB2_Temp.Values[39] := 0.0;
   BB2_Temp.Values[40] := 0.0;
   BB2_Temp.Values[41] := 0.0;
   BB2_Temp.Values[42] := 0.0;
   BB2_Temp.Values[43] := 0.0;
   BB2_Temp.Values[44] := 0.0;
   BB2_Temp.Values[45] := 0.0;
   BB2_Temp.Values[46] := 0.0;
   BB2_Temp.Values[47] := 0.0;
   BB2_Temp.Values[48] := 0.0;
   BB2_Temp.Values[49] := 0.0;
   BB2_Temp.Values[50] := 0.0;
   BB2_Temp.Values[51] := 0.0;
   BB2_Temp.Values[52] := 0.0;
   BB2_Temp.Values[53] := 0.0;
   BB2_Temp.Values[54] := 0.0;
   BB2_Temp.Values[55] := 0.0;
   BB2_Temp.Values[56] := 0.0;
   BB2_Temp.Values[57] := 0.0;
   BB2_Temp.Values[58] := 0.0;
   BB2_Temp.Values[59] := 0.0;
   BB2_Temp.Values[60] := 0.0;
   BB2_Temp.Values[61] := 0.0;
   BB2_Temp.Values[62] := 0.0;
   BB2_Temp.Values[63] := 0.0;
   BB2_Temp.Values[64] := 0.0;
   BB2_Temp.Values[65] := 0.0;
   BB2_Temp.Values[66] := 0.0;
   BB2_Temp.Values[67] := 0.0;
   BB2_Temp.Values[68] := 0.0;
   BB2_Temp.Values[69] := 0.0;
   BB2_Temp.Values[70] := 0.0;
   BB2_Temp.Values[71] := 0.0;
   BB2_Temp.Values[72] := 0.0;
   BB2_Temp.Values[73] := 0.0;
   BB2_Temp.Values[74] := 0.0;
   BB2_Temp.Values[75] := 0.0;
   BB2_Temp.Values[76] := 0.0;
   BB2_Temp.Values[77] := 0.0;
   BB2_Temp.Values[78] := 0.0;
   BB2_Temp.Values[79] := 0.0;
   BB2_Temp.Values[80] := 0.0;
   BB2_Temp.Values[81] := 0.0;
   BB2_Temp.Values[82] := 0.0;
   BB2_Temp.Values[83] := 0.0;
   BB2_Temp.Values[84] := 0.0;
   BB2_Temp.Values[85] := 0.0;
   BB2_Temp.Values[86] := 0.0;
   BB2_Temp.Values[87] := 0.0;
   BB2_Temp.Values[88] := 0.0;
   BB2_Temp.Values[89] := 0.0;
   BB2_Temp.Values[90] := 0.0;
   BB2_Temp.Values[91] := 0.0;
   BB2_Temp.Values[92] := 0.0;
   BB2_Temp.Values[93] := 0.0;
   BB2_Temp.Values[94] := 0.0;
   BB2_Temp.Values[95] := 0.0;
   BB2_Temp.Values[96] := 0.0;
   BB2_Temp.Values[97] := 0.0;
   BB2_Temp.Values[98] := 0.0;
   BB2_Temp.Values[99] := 0.0;
   BB2_Temp.Values[100] := 0.0;
   BB2_Temp.Values[101] := 0.0;
   BB2_Temp.Values[102] := 0.0;
   BB2_Temp.Values[103] := 0.0;
   BB2_Temp.Values[104] := 0.0;
   BB2_Temp.Values[105] := 0.0;
   BB2_Temp.Values[106] := 0.0;
   BB2_Temp.Values[107] := 0.0;
   BB2_Temp.Values[108] := 0.0;
   BB2_Temp.Values[109] := 0.0;
   BB2_Temp.Values[110] := 0.0;
   BB2_Temp.Values[111] := 0.0;
   BB2_Temp.Values[112] := 0.0;
   BB2_Temp.Values[113] := 0.0;
   BB2_Temp.Values[114] := 0.0;
   BB2_Temp.Values[115] := 0.0;
   BB2_Temp.Values[116] := 0.0;
   BB2_Temp.Values[117] := 0.0;
   BB2_Temp.Values[118] := 0.0;
   BB2_Temp.Values[119] := 0.0;
   BB1_DF.Values[0] := 0.0;
   BB1_DF.Values[1] := 0.0;
   BB1_DF.Values[2] := 0.0;
   BB1_DF.Values[3] := 0.0;
   BB1_DF.Values[4] := 0.0;
   BB1_DF.Values[5] := 0.0;
   BB1_DF.Values[6] := 0.0;
   BB1_DF.Values[7] := 0.0;
   BB1_DF.Values[8] := 0.0;
   BB1_DF.Values[9] := 0.0;
   BB1_DF.Values[10] := 0.0;
   BB1_DF.Values[11] := 0.0;
   BB1_DF.Values[12] := 0.0;
   BB1_DF.Values[13] := 0.0;
   BB1_DF.Values[14] := 0.0;
   BB1_DF.Values[15] := 0.0;
   BB1_DF.Values[16] := 0.0;
   BB1_DF.Values[17] := 0.0;
   BB1_DF.Values[18] := 0.0;
   BB1_DF.Values[19] := 0.0;
   BB1_DF.Values[20] := 0.0;
   BB1_DF.Values[21] := 0.0;
   BB1_DF.Values[22] := 0.0;
   BB1_DF.Values[23] := 0.0;
   BB1_DF.Values[24] := 0.0;
   BB1_DF.Values[25] := 0.0;
   BB1_DF.Values[26] := 0.0;
   BB1_DF.Values[27] := 0.0;
   BB1_DF.Values[28] := 0.0;
   BB1_DF.Values[29] := 0.0;
   BB1_DF.Values[30] := 0.0;
   BB1_DF.Values[31] := 0.0;
   BB1_DF.Values[32] := 0.0;
   BB1_DF.Values[33] := 0.0;
   BB1_DF.Values[34] := 0.0;
   BB1_DF.Values[35] := 0.0;
   BB1_DF.Values[36] := 0.0;
   BB1_DF.Values[37] := 0.0;
   BB1_DF.Values[38] := 0.0;
   BB1_DF.Values[39] := 0.0;
   BB1_DF.Values[40] := 0.0;
   BB1_DF.Values[41] := 0.0;
   BB1_DF.Values[42] := 0.0;
   BB1_DF.Values[43] := 0.0;
   BB1_DF.Values[44] := 0.0;
   BB1_DF.Values[45] := 0.0;
   BB1_DF.Values[46] := 0.0;
   BB1_DF.Values[47] := 0.0;
   BB1_DF.Values[48] := 0.0;
   BB1_DF.Values[49] := 0.0;
   BB1_DF.Values[50] := 0.0;
   BB1_DF.Values[51] := 0.0;
   BB1_DF.Values[52] := 0.0;
   BB1_DF.Values[53] := 0.0;
   BB1_DF.Values[54] := 0.0;
   BB1_DF.Values[55] := 0.0;
   BB1_DF.Values[56] := 0.0;
   BB1_DF.Values[57] := 0.0;
   BB1_DF.Values[58] := 0.0;
   BB1_DF.Values[59] := 0.0;
   BB1_DF.Values[60] := 0.0;
   BB1_DF.Values[61] := 0.0;
   BB1_DF.Values[62] := 0.0;
   BB1_DF.Values[63] := 0.0;
   BB1_DF.Values[64] := 0.0;
   BB1_DF.Values[65] := 0.0;
   BB1_DF.Values[66] := 0.0;
   BB1_DF.Values[67] := 0.0;
   BB1_DF.Values[68] := 0.0;
   BB1_DF.Values[69] := 0.0;
   BB1_DF.Values[70] := 0.0;
   BB1_DF.Values[71] := 0.0;
   BB1_DF.Values[72] := 0.0;
   BB1_DF.Values[73] := 0.0;
   BB1_DF.Values[74] := 0.0;
   BB1_DF.Values[75] := 0.0;
   BB1_DF.Values[76] := 0.0;
   BB1_DF.Values[77] := 0.0;
   BB1_DF.Values[78] := 0.0;
   BB1_DF.Values[79] := 0.0;
   BB1_DF.Values[80] := 0.0;
   BB1_DF.Values[81] := 0.0;
   BB1_DF.Values[82] := 0.0;
   BB1_DF.Values[83] := 0.0;
   BB1_DF.Values[84] := 0.0;
   BB1_DF.Values[85] := 0.0;
   BB1_DF.Values[86] := 0.0;
   BB1_DF.Values[87] := 0.0;
   BB1_DF.Values[88] := 0.0;
   BB1_DF.Values[89] := 0.0;
   BB1_DF.Values[90] := 0.0;
   BB1_DF.Values[91] := 0.0;
   BB1_DF.Values[92] := 0.0;
   BB1_DF.Values[93] := 0.0;
   BB1_DF.Values[94] := 0.0;
   BB1_DF.Values[95] := 0.0;
   BB1_DF.Values[96] := 0.0;
   BB1_DF.Values[97] := 0.0;
   BB1_DF.Values[98] := 0.0;
   BB1_DF.Values[99] := 0.0;
   BB1_DF.Values[100] := 0.0;
   BB1_DF.Values[101] := 0.0;
   BB1_DF.Values[102] := 0.0;
   BB1_DF.Values[103] := 0.0;
   BB1_DF.Values[104] := 0.0;
   BB1_DF.Values[105] := 0.0;
   BB1_DF.Values[106] := 0.0;
   BB1_DF.Values[107] := 0.0;
   BB1_DF.Values[108] := 0.0;
   BB1_DF.Values[109] := 0.0;
   BB1_DF.Values[110] := 0.0;
   BB1_DF.Values[111] := 0.0;
   BB1_DF.Values[112] := 0.0;
   BB1_DF.Values[113] := 0.0;
   BB1_DF.Values[114] := 0.0;
   BB1_DF.Values[115] := 0.0;
   BB1_DF.Values[116] := 0.0;
   BB1_DF.Values[117] := 0.0;
   BB1_DF.Values[118] := 0.0;
   BB1_DF.Values[119] := 0.0;
   BB2_DF.Values[0] := 0.0;
   BB2_DF.Values[1] := 0.0;
   BB2_DF.Values[2] := 0.0;
   BB2_DF.Values[3] := 0.0;
   BB2_DF.Values[4] := 0.0;
   BB2_DF.Values[5] := 0.0;
   BB2_DF.Values[6] := 0.0;
   BB2_DF.Values[7] := 0.0;
   BB2_DF.Values[8] := 0.0;
   BB2_DF.Values[9] := 0.0;
   BB2_DF.Values[10] := 19.97251;
   BB2_DF.Values[11] := 19.97251;
   BB2_DF.Values[12] := 19.97251;
   BB2_DF.Values[13] := 19.97251;
   BB2_DF.Values[14] := 19.97251;
   BB2_DF.Values[15] := 19.97251;
   BB2_DF.Values[16] := 19.97251;
   BB2_DF.Values[17] := 19.97251;
   BB2_DF.Values[18] := 19.97251;
   BB2_DF.Values[19] := 19.97251;
   BB2_DF.Values[20] := 19.97251;
   BB2_DF.Values[21] := 19.97251;
   BB2_DF.Values[22] := 19.97251;
   BB2_DF.Values[23] := 19.97251;
   BB2_DF.Values[24] := 19.97251;
   BB2_DF.Values[25] := 19.97251;
   BB2_DF.Values[26] := 19.97251;
   BB2_DF.Values[27] := 19.97251;
   BB2_DF.Values[28] := 19.97251;
   BB2_DF.Values[29] := 19.97251;
   BB2_DF.Values[30] := 0.0;
   BB2_DF.Values[31] := 0.0;
   BB2_DF.Values[32] := 0.0;
   BB2_DF.Values[33] := 0.0;
   BB2_DF.Values[34] := 0.0;
   BB2_DF.Values[35] := 0.0;
   BB2_DF.Values[36] := 0.0;
   BB2_DF.Values[37] := 0.0;
   BB2_DF.Values[38] := 0.0;
   BB2_DF.Values[39] := 0.0;
   BB2_DF.Values[40] := 0.0;
   BB2_DF.Values[41] := 0.0;
   BB2_DF.Values[42] := 0.0;
   BB2_DF.Values[43] := 0.0;
   BB2_DF.Values[44] := 0.0;
   BB2_DF.Values[45] := 0.0;
   BB2_DF.Values[46] := 0.0;
   BB2_DF.Values[47] := 0.0;
   BB2_DF.Values[48] := 0.0;
   BB2_DF.Values[49] := 0.0;
   BB2_DF.Values[50] := 0.0;
   BB2_DF.Values[51] := 0.0;
   BB2_DF.Values[52] := 0.0;
   BB2_DF.Values[53] := 0.0;
   BB2_DF.Values[54] := 0.0;
   BB2_DF.Values[55] := 0.0;
   BB2_DF.Values[56] := 0.0;
   BB2_DF.Values[57] := 0.0;
   BB2_DF.Values[58] := 0.0;
   BB2_DF.Values[59] := 0.0;
   BB2_DF.Values[60] := 0.0;
   BB2_DF.Values[61] := 0.0;
   BB2_DF.Values[62] := 0.0;
   BB2_DF.Values[63] := 0.0;
   BB2_DF.Values[64] := 0.0;
   BB2_DF.Values[65] := 0.0;
   BB2_DF.Values[66] := 0.0;
   BB2_DF.Values[67] := 0.0;
   BB2_DF.Values[68] := 0.0;
   BB2_DF.Values[69] := 0.0;
   BB2_DF.Values[70] := 0.0;
   BB2_DF.Values[71] := 0.0;
   BB2_DF.Values[72] := 0.0;
   BB2_DF.Values[73] := 0.0;
   BB2_DF.Values[74] := 0.0;
   BB2_DF.Values[75] := 0.0;
   BB2_DF.Values[76] := 0.0;
   BB2_DF.Values[77] := 0.0;
   BB2_DF.Values[78] := 0.0;
   BB2_DF.Values[79] := 0.0;
   BB2_DF.Values[80] := 0.0;
   BB2_DF.Values[81] := 0.0;
   BB2_DF.Values[82] := 0.0;
   BB2_DF.Values[83] := 0.0;
   BB2_DF.Values[84] := 0.0;
   BB2_DF.Values[85] := 0.0;
   BB2_DF.Values[86] := 0.0;
   BB2_DF.Values[87] := 0.0;
   BB2_DF.Values[88] := 0.0;
   BB2_DF.Values[89] := 0.0;
   BB2_DF.Values[90] := 0.0;
   BB2_DF.Values[91] := 0.0;
   BB2_DF.Values[92] := 0.0;
   BB2_DF.Values[93] := 0.0;
   BB2_DF.Values[94] := 0.0;
   BB2_DF.Values[95] := 0.0;
   BB2_DF.Values[96] := 0.0;
   BB2_DF.Values[97] := 0.0;
   BB2_DF.Values[98] := 0.0;
   BB2_DF.Values[99] := 0.0;
   BB2_DF.Values[100] := 0.0;
   BB2_DF.Values[101] := 0.0;
   BB2_DF.Values[102] := 0.0;
   BB2_DF.Values[103] := 0.0;
   BB2_DF.Values[104] := 0.0;
   BB2_DF.Values[105] := 0.0;
   BB2_DF.Values[106] := 0.0;
   BB2_DF.Values[107] := 0.0;
   BB2_DF.Values[108] := 0.0;
   BB2_DF.Values[109] := 0.0;
   BB2_DF.Values[110] := 0.0;
   BB2_DF.Values[111] := 0.0;
   BB2_DF.Values[112] := 0.0;
   BB2_DF.Values[113] := 0.0;
   BB2_DF.Values[114] := 0.0;
   BB2_DF.Values[115] := 0.0;
   BB2_DF.Values[116] := 0.0;
   BB2_DF.Values[117] := 0.0;
   BB2_DF.Values[118] := 0.0;
   BB2_DF.Values[119] := 0.0;
   Zulauf_Niv.Values[0] := 0.262218;
   Zulauf_Niv.Values[1] := 0.899679;
   Zulauf_Niv.Values[2] := 2.206248;
   Zulauf_Niv.Values[3] := 2.816583;
   Zulauf_Niv.Values[4] := 3.820245;
   Zulauf_Niv.Values[5] := 4.909806;
   Zulauf_Niv.Values[6] := 5.393553;
   Zulauf_Niv.Values[7] := 0.257697;
   Zulauf_Niv.Values[8] := 0.266739;
   Zulauf_Niv.Values[9] := 0.262218;
   Zulauf_Niv.Values[10] := 0.0101053;
   Zulauf_Niv.Values[11] := 0.0101053;
   Zulauf_Niv.Values[12] := 0.0101053;
   Zulauf_Niv.Values[13] := 0.0101053;
   Zulauf_Niv.Values[14] := 0.0101053;
   Zulauf_Niv.Values[15] := 0.0101053;
   Zulauf_Niv.Values[16] := 0.0101053;
   Zulauf_Niv.Values[17] := 0.0101053;
   Zulauf_Niv.Values[18] := 0.0101053;
   Zulauf_Niv.Values[19] := 0.0101053;
   Zulauf_Niv.Values[20] := 0.0101053;
   Zulauf_Niv.Values[21] := 0.0101053;
   Zulauf_Niv.Values[22] := 0.0101053;
   Zulauf_Niv.Values[23] := 0.0101053;
   Zulauf_Niv.Values[24] := 0.0101053;
   Zulauf_Niv.Values[25] := 0.0101053;
   Zulauf_Niv.Values[26] := 0.0101053;
   Zulauf_Niv.Values[27] := 0.0101053;
   Zulauf_Niv.Values[28] := 0.0101053;
   Zulauf_Niv.Values[29] := 0.0101053;
   Zulauf_Niv.Values[30] := 0.0;
   Zulauf_Niv.Values[31] := 0.0;
   Zulauf_Niv.Values[32] := 0.0;
   Zulauf_Niv.Values[33] := 0.0;
   Zulauf_Niv.Values[34] := 0.0;
   Zulauf_Niv.Values[35] := 0.0;
   Zulauf_Niv.Values[36] := 0.0;
   Zulauf_Niv.Values[37] := 0.0;
   Zulauf_Niv.Values[38] := 0.0;
   Zulauf_Niv.Values[39] := 0.0;
   Zulauf_Niv.Values[40] := 0.0;
   Zulauf_Niv.Values[41] := 0.0;
   Zulauf_Niv.Values[42] := 0.0;
   Zulauf_Niv.Values[43] := 0.0;
   Zulauf_Niv.Values[44] := 0.0;
   Zulauf_Niv.Values[45] := 0.0;
   Zulauf_Niv.Values[46] := 0.0;
   Zulauf_Niv.Values[47] := 0.0;
   Zulauf_Niv.Values[48] := 0.0;
   Zulauf_Niv.Values[49] := 0.0;
   Zulauf_Niv.Values[50] := 0.0;
   Zulauf_Niv.Values[51] := 0.0;
   Zulauf_Niv.Values[52] := 0.0;
   Zulauf_Niv.Values[53] := 0.0;
   Zulauf_Niv.Values[54] := 0.0;
   Zulauf_Niv.Values[55] := 0.0;
   Zulauf_Niv.Values[56] := 0.0;
   Zulauf_Niv.Values[57] := 0.0;
   Zulauf_Niv.Values[58] := 0.0;
   Zulauf_Niv.Values[59] := 0.0;
   Zulauf_Niv.Values[60] := 0.0;
   Zulauf_Niv.Values[61] := 0.0;
   Zulauf_Niv.Values[62] := 0.0;
   Zulauf_Niv.Values[63] := 0.0;
   Zulauf_Niv.Values[64] := 0.0;
   Zulauf_Niv.Values[65] := 0.0;
   Zulauf_Niv.Values[66] := 0.0;
   Zulauf_Niv.Values[67] := 0.0;
   Zulauf_Niv.Values[68] := 0.0;
   Zulauf_Niv.Values[69] := 0.0;
   Zulauf_Niv.Values[70] := 0.0;
   Zulauf_Niv.Values[71] := 0.0;
   Zulauf_Niv.Values[72] := 0.0;
   Zulauf_Niv.Values[73] := 0.0;
   Zulauf_Niv.Values[74] := 0.0;
   Zulauf_Niv.Values[75] := 0.0;
   Zulauf_Niv.Values[76] := 0.0;
   Zulauf_Niv.Values[77] := 0.0;
   Zulauf_Niv.Values[78] := 0.0;
   Zulauf_Niv.Values[79] := 0.0;
   Zulauf_Niv.Values[80] := 0.0;
   Zulauf_Niv.Values[81] := 0.0;
   Zulauf_Niv.Values[82] := 0.0;
   Zulauf_Niv.Values[83] := 0.0;
   Zulauf_Niv.Values[84] := 0.0;
   Zulauf_Niv.Values[85] := 0.0;
   Zulauf_Niv.Values[86] := 0.0;
   Zulauf_Niv.Values[87] := 0.0;
   Zulauf_Niv.Values[88] := 0.0;
   Zulauf_Niv.Values[89] := 0.0;
   Zulauf_Niv.Values[90] := 0.0;
   Zulauf_Niv.Values[91] := 0.0;
   Zulauf_Niv.Values[92] := 0.0;
   Zulauf_Niv.Values[93] := 0.0;
   Zulauf_Niv.Values[94] := 0.0;
   Zulauf_Niv.Values[95] := 0.0;
   Zulauf_Niv.Values[96] := 0.0;
   Zulauf_Niv.Values[97] := 0.0;
   Zulauf_Niv.Values[98] := 0.0;
   Zulauf_Niv.Values[99] := 0.0;
   Zulauf_Niv.Values[100] := 0.0;
   Zulauf_Niv.Values[101] := 0.0;
   Zulauf_Niv.Values[102] := 0.0;
   Zulauf_Niv.Values[103] := 0.0;
   Zulauf_Niv.Values[104] := 0.0;
   Zulauf_Niv.Values[105] := 0.0;
   Zulauf_Niv.Values[106] := 0.0;
   Zulauf_Niv.Values[107] := 0.0;
   Zulauf_Niv.Values[108] := 0.0;
   Zulauf_Niv.Values[109] := 0.0;
   Zulauf_Niv.Values[110] := 0.0;
   Zulauf_Niv.Values[111] := 0.0;
   Zulauf_Niv.Values[112] := 0.0;
   Zulauf_Niv.Values[113] := 0.0;
   Zulauf_Niv.Values[114] := 0.0;
   Zulauf_Niv.Values[115] := 0.0;
   Zulauf_Niv.Values[116] := 0.0;
   Zulauf_Niv.Values[117] := 0.0;
   Zulauf_Niv.Values[118] := 0.0;
   Zulauf_Niv.Values[119] := 0.0;
   Zulauf_DF.Values[0] := -0.0067815;
   Zulauf_DF.Values[1] := -0.0067815;
   Zulauf_DF.Values[2] := -0.0067815;
   Zulauf_DF.Values[3] := -0.0067815;
   Zulauf_DF.Values[4] := -0.0067815;
   Zulauf_DF.Values[5] := -0.0067815;
   Zulauf_DF.Values[6] := -0.0067815;
   Zulauf_DF.Values[7] := -0.0067815;
   Zulauf_DF.Values[8] := -0.009042;
   Zulauf_DF.Values[9] := -0.009042;
   Zulauf_DF.Values[10] := 0.0;
   Zulauf_DF.Values[11] := 0.0;
   Zulauf_DF.Values[12] := 0.0;
   Zulauf_DF.Values[13] := 0.0;
   Zulauf_DF.Values[14] := 0.0;
   Zulauf_DF.Values[15] := 0.0;
   Zulauf_DF.Values[16] := 0.0;
   Zulauf_DF.Values[17] := 0.0;
   Zulauf_DF.Values[18] := 0.0;
   Zulauf_DF.Values[19] := 0.0;
   Zulauf_DF.Values[20] := 0.0;
   Zulauf_DF.Values[21] := 0.0;
   Zulauf_DF.Values[22] := 0.0;
   Zulauf_DF.Values[23] := 0.0;
   Zulauf_DF.Values[24] := 0.0;
   Zulauf_DF.Values[25] := 0.0;
   Zulauf_DF.Values[26] := 0.0;
   Zulauf_DF.Values[27] := 0.0;
   Zulauf_DF.Values[28] := 0.0;
   Zulauf_DF.Values[29] := 0.0;
   Zulauf_DF.Values[30] := 0.0;
   Zulauf_DF.Values[31] := 0.0;
   Zulauf_DF.Values[32] := 0.0;
   Zulauf_DF.Values[33] := 0.0;
   Zulauf_DF.Values[34] := 0.0;
   Zulauf_DF.Values[35] := 0.0;
   Zulauf_DF.Values[36] := 0.0;
   Zulauf_DF.Values[37] := 0.0;
   Zulauf_DF.Values[38] := 0.0;
   Zulauf_DF.Values[39] := 0.0;
   Zulauf_DF.Values[40] := 0.0;
   Zulauf_DF.Values[41] := 0.0;
   Zulauf_DF.Values[42] := 0.0;
   Zulauf_DF.Values[43] := 0.0;
   Zulauf_DF.Values[44] := 0.0;
   Zulauf_DF.Values[45] := 0.0;
   Zulauf_DF.Values[46] := 0.0;
   Zulauf_DF.Values[47] := 0.0;
   Zulauf_DF.Values[48] := 0.0;
   Zulauf_DF.Values[49] := 0.0;
   Zulauf_DF.Values[50] := 0.0;
   Zulauf_DF.Values[51] := 0.0;
   Zulauf_DF.Values[52] := 0.0;
   Zulauf_DF.Values[53] := 0.0;
   Zulauf_DF.Values[54] := 0.0;
   Zulauf_DF.Values[55] := 0.0;
   Zulauf_DF.Values[56] := 0.0;
   Zulauf_DF.Values[57] := 0.0;
   Zulauf_DF.Values[58] := 0.0;
   Zulauf_DF.Values[59] := 0.0;
   Zulauf_DF.Values[60] := 0.0;
   Zulauf_DF.Values[61] := 0.0;
   Zulauf_DF.Values[62] := 0.0;
   Zulauf_DF.Values[63] := 0.0;
   Zulauf_DF.Values[64] := 0.0;
   Zulauf_DF.Values[65] := 0.0;
   Zulauf_DF.Values[66] := 0.0;
   Zulauf_DF.Values[67] := 0.0;
   Zulauf_DF.Values[68] := 0.0;
   Zulauf_DF.Values[69] := 0.0;
   Zulauf_DF.Values[70] := 0.0;
   Zulauf_DF.Values[71] := 0.0;
   Zulauf_DF.Values[72] := 0.0;
   Zulauf_DF.Values[73] := 0.0;
   Zulauf_DF.Values[74] := 0.0;
   Zulauf_DF.Values[75] := 0.0;
   Zulauf_DF.Values[76] := 0.0;
   Zulauf_DF.Values[77] := 0.0;
   Zulauf_DF.Values[78] := 0.0;
   Zulauf_DF.Values[79] := 0.0;
   Zulauf_DF.Values[80] := 0.0;
   Zulauf_DF.Values[81] := 0.0;
   Zulauf_DF.Values[82] := 0.0;
   Zulauf_DF.Values[83] := 0.0;
   Zulauf_DF.Values[84] := 0.0;
   Zulauf_DF.Values[85] := 0.0;
   Zulauf_DF.Values[86] := 0.0;
   Zulauf_DF.Values[87] := 0.0;
   Zulauf_DF.Values[88] := 0.0;
   Zulauf_DF.Values[89] := 0.0;
   Zulauf_DF.Values[90] := 0.0;
   Zulauf_DF.Values[91] := 0.0;
   Zulauf_DF.Values[92] := 0.0;
   Zulauf_DF.Values[93] := 0.0;
   Zulauf_DF.Values[94] := 0.0;
   Zulauf_DF.Values[95] := 0.0;
   Zulauf_DF.Values[96] := 0.0;
   Zulauf_DF.Values[97] := 0.0;
   Zulauf_DF.Values[98] := 0.0;
   Zulauf_DF.Values[99] := 0.0;
   Zulauf_DF.Values[100] := 0.0;
   Zulauf_DF.Values[101] := 0.0;
   Zulauf_DF.Values[102] := 0.0;
   Zulauf_DF.Values[103] := 0.0;
   Zulauf_DF.Values[104] := 0.0;
   Zulauf_DF.Values[105] := 0.0;
   Zulauf_DF.Values[106] := 0.0;
   Zulauf_DF.Values[107] := 0.0;
   Zulauf_DF.Values[108] := 0.0;
   Zulauf_DF.Values[109] := 0.0;
   Zulauf_DF.Values[110] := 0.0;
   Zulauf_DF.Values[111] := 0.0;
   Zulauf_DF.Values[112] := 0.0;
   Zulauf_DF.Values[113] := 0.0;
   Zulauf_DF.Values[114] := 0.0;
   Zulauf_DF.Values[115] := 0.0;
   Zulauf_DF.Values[116] := 0.0;
   Zulauf_DF.Values[117] := 0.0;
   Zulauf_DF.Values[118] := 0.0;
   Zulauf_DF.Values[119] := 0.0;
   Verteiler_pH.Values[0] := 2.0;
   Verteiler_pH.Values[1] := 2.0;
   Verteiler_pH.Values[2] := 2.0;
   Verteiler_pH.Values[3] := 2.0;
   Verteiler_pH.Values[4] := 2.0;
   Verteiler_pH.Values[5] := 2.0;
   Verteiler_pH.Values[6] := 2.0;
   Verteiler_pH.Values[7] := 2.0;
   Verteiler_pH.Values[8] := 2.0;
   Verteiler_pH.Values[9] := 2.0;
   Verteiler_pH.Values[10] := 0.0;
   Verteiler_pH.Values[11] := 0.0;
   Verteiler_pH.Values[12] := 0.0;
   Verteiler_pH.Values[13] := 0.0;
   Verteiler_pH.Values[14] := 0.0;
   Verteiler_pH.Values[15] := 0.0;
   Verteiler_pH.Values[16] := 0.0;
   Verteiler_pH.Values[17] := 0.0;
   Verteiler_pH.Values[18] := 0.0;
   Verteiler_pH.Values[19] := 0.0;
   Verteiler_pH.Values[20] := 0.0;
   Verteiler_pH.Values[21] := 0.0;
   Verteiler_pH.Values[22] := 0.0;
   Verteiler_pH.Values[23] := 0.0;
   Verteiler_pH.Values[24] := 0.0;
   Verteiler_pH.Values[25] := 0.0;
   Verteiler_pH.Values[26] := 0.0;
   Verteiler_pH.Values[27] := 0.0;
   Verteiler_pH.Values[28] := 0.0;
   Verteiler_pH.Values[29] := 0.0;
   Verteiler_pH.Values[30] := 0.0;
   Verteiler_pH.Values[31] := 0.0;
   Verteiler_pH.Values[32] := 0.0;
   Verteiler_pH.Values[33] := 0.0;
   Verteiler_pH.Values[34] := 0.0;
   Verteiler_pH.Values[35] := 0.0;
   Verteiler_pH.Values[36] := 0.0;
   Verteiler_pH.Values[37] := 0.0;
   Verteiler_pH.Values[38] := 0.0;
   Verteiler_pH.Values[39] := 0.0;
   Verteiler_pH.Values[40] := 0.0;
   Verteiler_pH.Values[41] := 0.0;
   Verteiler_pH.Values[42] := 0.0;
   Verteiler_pH.Values[43] := 0.0;
   Verteiler_pH.Values[44] := 0.0;
   Verteiler_pH.Values[45] := 0.0;
   Verteiler_pH.Values[46] := 0.0;
   Verteiler_pH.Values[47] := 0.0;
   Verteiler_pH.Values[48] := 0.0;
   Verteiler_pH.Values[49] := 0.0;
   Verteiler_pH.Values[50] := 0.0;
   Verteiler_pH.Values[51] := 0.0;
   Verteiler_pH.Values[52] := 0.0;
   Verteiler_pH.Values[53] := 0.0;
   Verteiler_pH.Values[54] := 0.0;
   Verteiler_pH.Values[55] := 0.0;
   Verteiler_pH.Values[56] := 0.0;
   Verteiler_pH.Values[57] := 0.0;
   Verteiler_pH.Values[58] := 0.0;
   Verteiler_pH.Values[59] := 0.0;
   Verteiler_pH.Values[60] := 0.0;
   Verteiler_pH.Values[61] := 0.0;
   Verteiler_pH.Values[62] := 0.0;
   Verteiler_pH.Values[63] := 0.0;
   Verteiler_pH.Values[64] := 0.0;
   Verteiler_pH.Values[65] := 0.0;
   Verteiler_pH.Values[66] := 0.0;
   Verteiler_pH.Values[67] := 0.0;
   Verteiler_pH.Values[68] := 0.0;
   Verteiler_pH.Values[69] := 0.0;
   Verteiler_pH.Values[70] := 0.0;
   Verteiler_pH.Values[71] := 0.0;
   Verteiler_pH.Values[72] := 0.0;
   Verteiler_pH.Values[73] := 0.0;
   Verteiler_pH.Values[74] := 0.0;
   Verteiler_pH.Values[75] := 0.0;
   Verteiler_pH.Values[76] := 0.0;
   Verteiler_pH.Values[77] := 0.0;
   Verteiler_pH.Values[78] := 0.0;
   Verteiler_pH.Values[79] := 0.0;
   Verteiler_pH.Values[80] := 0.0;
   Verteiler_pH.Values[81] := 0.0;
   Verteiler_pH.Values[82] := 0.0;
   Verteiler_pH.Values[83] := 0.0;
   Verteiler_pH.Values[84] := 0.0;
   Verteiler_pH.Values[85] := 0.0;
   Verteiler_pH.Values[86] := 0.0;
   Verteiler_pH.Values[87] := 0.0;
   Verteiler_pH.Values[88] := 0.0;
   Verteiler_pH.Values[89] := 0.0;
   Verteiler_pH.Values[90] := 0.0;
   Verteiler_pH.Values[91] := 0.0;
   Verteiler_pH.Values[92] := 0.0;
   Verteiler_pH.Values[93] := 0.0;
   Verteiler_pH.Values[94] := 0.0;
   Verteiler_pH.Values[95] := 0.0;
   Verteiler_pH.Values[96] := 0.0;
   Verteiler_pH.Values[97] := 0.0;
   Verteiler_pH.Values[98] := 0.0;
   Verteiler_pH.Values[99] := 0.0;
   Verteiler_pH.Values[100] := 0.0;
   Verteiler_pH.Values[101] := 0.0;
   Verteiler_pH.Values[102] := 0.0;
   Verteiler_pH.Values[103] := 0.0;
   Verteiler_pH.Values[104] := 0.0;
   Verteiler_pH.Values[105] := 0.0;
   Verteiler_pH.Values[106] := 0.0;
   Verteiler_pH.Values[107] := 0.0;
   Verteiler_pH.Values[108] := 0.0;
   Verteiler_pH.Values[109] := 0.0;
   Verteiler_pH.Values[110] := 0.0;
   Verteiler_pH.Values[111] := 0.0;
   Verteiler_pH.Values[112] := 0.0;
   Verteiler_pH.Values[113] := 0.0;
   Verteiler_pH.Values[114] := 0.0;
   Verteiler_pH.Values[115] := 0.0;
   Verteiler_pH.Values[116] := 0.0;
   Verteiler_pH.Values[117] := 0.0;
   Verteiler_pH.Values[118] := 0.0;
   Verteiler_pH.Values[119] := 0.0;
   Verteiler_O2.Values[0] := 0.0;
   Verteiler_O2.Values[1] := 0.0;
   Verteiler_O2.Values[2] := 0.0;
   Verteiler_O2.Values[3] := 0.0;
   Verteiler_O2.Values[4] := 0.0;
   Verteiler_O2.Values[5] := 0.0;
   Verteiler_O2.Values[6] := 0.0;
   Verteiler_O2.Values[7] := 0.0;
   Verteiler_O2.Values[8] := 0.0;
   Verteiler_O2.Values[9] := 0.0;
   Verteiler_O2.Values[10] := 0.0;
   Verteiler_O2.Values[11] := 0.0;
   Verteiler_O2.Values[12] := 0.0;
   Verteiler_O2.Values[13] := 0.0;
   Verteiler_O2.Values[14] := 0.0;
   Verteiler_O2.Values[15] := 0.0;
   Verteiler_O2.Values[16] := 0.0;
   Verteiler_O2.Values[17] := 0.0;
   Verteiler_O2.Values[18] := 0.0;
   Verteiler_O2.Values[19] := 0.0;
   Verteiler_O2.Values[20] := 2.48256;
   Verteiler_O2.Values[21] := 2.48256;
   Verteiler_O2.Values[22] := 2.48256;
   Verteiler_O2.Values[23] := 2.48256;
   Verteiler_O2.Values[24] := 2.48256;
   Verteiler_O2.Values[25] := 2.48256;
   Verteiler_O2.Values[26] := 2.48256;
   Verteiler_O2.Values[27] := 2.48256;
   Verteiler_O2.Values[28] := 2.48256;
   Verteiler_O2.Values[29] := 2.48256;
   Verteiler_O2.Values[30] := 0.0;
   Verteiler_O2.Values[31] := 0.0;
   Verteiler_O2.Values[32] := 0.0;
   Verteiler_O2.Values[33] := 0.0;
   Verteiler_O2.Values[34] := 0.0;
   Verteiler_O2.Values[35] := 0.0;
   Verteiler_O2.Values[36] := 0.0;
   Verteiler_O2.Values[37] := 0.0;
   Verteiler_O2.Values[38] := 0.0;
   Verteiler_O2.Values[39] := 0.0;
   Verteiler_O2.Values[40] := 0.0;
   Verteiler_O2.Values[41] := 0.0;
   Verteiler_O2.Values[42] := 0.0;
   Verteiler_O2.Values[43] := 0.0;
   Verteiler_O2.Values[44] := 0.0;
   Verteiler_O2.Values[45] := 0.0;
   Verteiler_O2.Values[46] := 0.0;
   Verteiler_O2.Values[47] := 0.0;
   Verteiler_O2.Values[48] := 0.0;
   Verteiler_O2.Values[49] := 0.0;
   Verteiler_O2.Values[50] := 0.0;
   Verteiler_O2.Values[51] := 0.0;
   Verteiler_O2.Values[52] := 0.0;
   Verteiler_O2.Values[53] := 0.0;
   Verteiler_O2.Values[54] := 0.0;
   Verteiler_O2.Values[55] := 0.0;
   Verteiler_O2.Values[56] := 0.0;
   Verteiler_O2.Values[57] := 0.0;
   Verteiler_O2.Values[58] := 0.0;
   Verteiler_O2.Values[59] := 0.0;
   Verteiler_O2.Values[60] := 0.0;
   Verteiler_O2.Values[61] := 0.0;
   Verteiler_O2.Values[62] := 0.0;
   Verteiler_O2.Values[63] := 0.0;
   Verteiler_O2.Values[64] := 0.0;
   Verteiler_O2.Values[65] := 0.0;
   Verteiler_O2.Values[66] := 0.0;
   Verteiler_O2.Values[67] := 0.0;
   Verteiler_O2.Values[68] := 0.0;
   Verteiler_O2.Values[69] := 0.0;
   Verteiler_O2.Values[70] := 0.0;
   Verteiler_O2.Values[71] := 0.0;
   Verteiler_O2.Values[72] := 0.0;
   Verteiler_O2.Values[73] := 0.0;
   Verteiler_O2.Values[74] := 0.0;
   Verteiler_O2.Values[75] := 0.0;
   Verteiler_O2.Values[76] := 0.0;
   Verteiler_O2.Values[77] := 0.0;
   Verteiler_O2.Values[78] := 0.0;
   Verteiler_O2.Values[79] := 0.0;
   Verteiler_O2.Values[80] := 0.0;
   Verteiler_O2.Values[81] := 0.0;
   Verteiler_O2.Values[82] := 0.0;
   Verteiler_O2.Values[83] := 0.0;
   Verteiler_O2.Values[84] := 0.0;
   Verteiler_O2.Values[85] := 0.0;
   Verteiler_O2.Values[86] := 0.0;
   Verteiler_O2.Values[87] := 0.0;
   Verteiler_O2.Values[88] := 0.0;
   Verteiler_O2.Values[89] := 0.0;
   Verteiler_O2.Values[90] := 0.0;
   Verteiler_O2.Values[91] := 0.0;
   Verteiler_O2.Values[92] := 0.0;
   Verteiler_O2.Values[93] := 0.0;
   Verteiler_O2.Values[94] := 0.0;
   Verteiler_O2.Values[95] := 0.0;
   Verteiler_O2.Values[96] := 0.0;
   Verteiler_O2.Values[97] := 0.0;
   Verteiler_O2.Values[98] := 0.0;
   Verteiler_O2.Values[99] := 0.0;
   Verteiler_O2.Values[100] := 0.0;
   Verteiler_O2.Values[101] := 0.0;
   Verteiler_O2.Values[102] := 0.0;
   Verteiler_O2.Values[103] := 0.0;
   Verteiler_O2.Values[104] := 0.0;
   Verteiler_O2.Values[105] := 0.0;
